SPLINE
SPL {X  -165.650, Y  +556.469, Z    +0.000, E1   +47.823, E3 +319681.375}
SPL {X  -165.650, Y  +549.545, Z    +0.000, E1   +47.953, E3 +319693.501}
SPL {X  -165.650, Y  +541.974, Z    +0.000, E1   +47.882, E3 +319707.890}
SPL {X  -165.650, Y  +535.023, Z    +0.000, E1   +47.697, E3 +319721.879}
SPL {X  -165.650, Y  +526.169, Z    +0.000, E1   +47.853, E3 +319737.474}
SPL {X  -165.650, Y  +520.016, Z    +0.000, E1   +47.658, E3 +319749.858}
SPL {X  -165.650, Y  +512.416, Z    +0.000, E1   +48.035, E3 +319761.825}
SPL {X  -165.650, Y  +507.257, Z    +0.000, E1   +47.748, E3 +319772.892}
SPL {X  -165.650, Y  +501.812, Z    +0.000, E1   +47.738, E3 +319783.175}
SPL {X  -165.650, Y  +493.465, Z    +0.000, E1   +47.959, E3 +319797.346}
SPL {X  -165.650, Y  +486.149, Z    +0.000, E1   +47.831, E3 +319811.621}
SPL {X  -165.650, Y  +479.821, Z    +0.000, E1   +47.727, E3 +319823.895}
SPL {X  -165.650, Y  +472.739, Z    +0.000, E1   +47.923, E3 +319835.914}
SPL {X  -165.650, Y  +466.586, Z    +0.000, E1   +48.125, E3 +319845.928}
SPL {X  -165.650, Y  +464.575, Z    +0.000, E1   +47.451, E3 +319853.694}
SPL {X  -165.650, Y  +456.851, Z    +0.000, E1   +47.856, E3 +319865.800}
SPL {X  -165.650, Y  +449.262, Z    +0.000, E1   +48.080, E3 +319878.366}
SPL {X  -165.650, Y  +436.765, Z    +0.000, E1   +49.819, E3 +319890.265}
SPL {X  -165.650, Y  +430.891, Z    +0.000, E1   +49.130, E3 +319904.767}
SPL {X  -165.650, Y  +423.272, Z    +0.000, E1   +49.176, E3 +319917.805}
SPL {X  -165.650, Y  +416.522, Z    +0.000, E1   +49.338, E3 +319928.783}
SPL {X  -165.650, Y  +410.777, Z    +0.000, E1   +49.173, E3 +319939.835}
SPL {X  -165.650, Y  +405.230, Z    +0.000, E1   +49.266, E3 +319949.038}
SPL {X  -165.650, Y  +398.850, Z    +0.000, E1   +49.279, E3 +319960.330}
SPL {X  -165.650, Y  +391.803, Z    +0.000, E1   +49.319, E3 +319972.367}
SPL {X  -165.650, Y  +386.526, Z    +0.000, E1   +49.193, E3 +319982.457}
SPL {X  -165.650, Y  +381.684, Z    +0.000, E1   +49.061, E3 +319991.742}
SPL {X  -165.602, Y  +374.507, Z    +0.000, E1   +49.269, E3 +320003.334}
SPL {X  -165.183, Y  +366.070, Z    +0.000, E1   +49.261, E3 +320018.218}
SPL {X  -164.692, Y  +360.715, Z    +0.000, E1   +48.960, E3 +320029.299}
SPL {X  -163.908, Y  +354.543, Z    +0.000, E1   +49.169, E3 +320038.990}
SPL {X  -163.052, Y  +349.277, Z    +0.000, E1   +48.680, E3 +320051.095}
SPL {X  -162.125, Y  +344.507, Z    +0.000, E1   +48.543, E3 +320060.235}
SPL {X  -160.947, Y  +339.310, Z    +0.000, E1   +48.561, E3 +320069.344}
SPL {X  -159.860, Y  +335.086, Z    +0.000, E1   +48.145, E3 +320079.056}
SPL {X  -158.277, Y  +329.631, Z    +0.000, E1   +47.981, E3 +320089.678}
SPL {X  -156.804, Y  +325.092, Z    +0.000, E1   +47.609, E3 +320099.571}
SPL {X  -155.465, Y  +321.311, Z    +0.000, E1   +47.446, E3 +320107.106}
SPL {X  -153.706, Y  +316.739, Z    +0.000, E1   +47.523, E3 +320114.719}
SPL {X  -143.727, Y  +296.145, Z    +0.000, E1   +53.260, E3 +320117.863}
SPL {X  -128.440, Y  +273.891, Z    +0.000, E1   +47.966, E3 +320205.109}
ENDSPLINE

SPLINE
SPL {X  -131.798, Y  +278.155, Z    +0.000, E1   +45.574, E3 +320230.736}
SPL {X  -154.181, Y  +317.936, Z    +0.000, E1   +32.662, E3 +320296.072}
SPL {X  -162.537, Y  +346.536, Z    +0.000, E1   +20.123, E3 +320295.293}
SPL {X  -164.610, Y  +359.970, Z    +0.000, E1   +13.118, E3 +320290.159}
SPL {X  -165.367, Y  +368.828, Z    +0.000, E1    +8.137, E3 +320288.612}
SPL {X  -165.621, Y  +375.422, Z    +0.000, E1    +4.067, E3 +320289.489}
SPL {X  -165.650, Y  +379.733, Z    +0.000, E1    +1.160, E3 +320287.795}
SPL {X  -165.650, Y  +383.552, Z    +0.000, E1    -1.868, E3 +320287.045}
SPL {X  -165.650, Y  +387.323, Z    +0.000, E1    -5.609, E3 +320286.861}
SPL {X  -165.650, Y  +392.013, Z    +0.000, E1   -10.856, E3 +320285.878}
SPL {X  -165.650, Y  +398.769, Z    +0.000, E1   -19.304, E3 +320284.490}
SPL {X  -165.650, Y  +407.471, Z    +0.000, E1   -31.017, E3 +320280.648}
SPL {X  -165.650, Y  +414.706, Z    +0.000, E1   -39.242, E3 +320279.624}
SPL {X  -165.650, Y  +446.037, Z    +0.000, E1   -53.739, E3 +320294.230}
SPL {X  -165.650, Y  +454.158, Z    +0.000, E1   -53.343, E3 +320304.582}
SPL {X  -165.650, Y  +513.780, Z    +0.000, E1   -56.183, E3 +320365.379}
ENDSPLINE

SPLINE
SPL {X  -165.650, Y  +495.869, Z    +0.000, E1   -48.812, E3 +320381.567}
ENDSPLINE

SPLINE
SPL {X  -165.650, Y  +504.906, Z    +0.000, E1   -48.979, E3 +320396.887}
SPL {X  -165.650, Y  +512.952, Z    +0.000, E1   -48.898, E3 +320411.509}
SPL {X  -165.650, Y  +519.321, Z    +0.000, E1   -49.041, E3 +320421.977}
SPL {X  -165.650, Y  +524.312, Z    +0.000, E1   -48.855, E3 +320432.002}
SPL {X  -165.650, Y  +530.631, Z    +0.000, E1   -48.990, E3 +320442.462}
SPL {X  -165.650, Y  +536.725, Z    +0.000, E1   -48.843, E3 +320454.213}
SPL {X  -165.650, Y  +542.959, Z    +0.000, E1   -48.923, E3 +320464.828}
SPL {X  -165.650, Y  +548.939, Z    +0.000, E1   -48.968, E3 +320475.222}
SPL {X  -165.650, Y  +553.607, Z    +0.000, E1   -48.716, E3 +320485.040}
SPL {X  -165.650, Y  +562.368, Z    +0.000, E1   -49.014, E3 +320499.100}
SPL {X  -165.650, Y  +570.317, Z    +0.000, E1   -48.893, E3 +320513.843}
SPL {X  -165.650, Y  +577.487, Z    +0.000, E1   -49.001, E3 +320525.951}
SPL {X  -165.650, Y  +581.837, Z    +0.000, E1   -48.612, E3 +320535.984}
SPL {X  -165.650, Y  +588.614, Z    +0.000, E1   -49.053, E3 +320545.502}
SPL {X  -165.650, Y  +593.784, Z    +0.000, E1   -48.711, E3 +320556.787}
SPL {X  -165.650, Y  +600.281, Z    +0.000, E1   -48.957, E3 +320566.890}
SPL {X  -165.650, Y  +606.252, Z    +0.000, E1   -48.984, E3 +320577.423}
SPL {X  -165.650, Y  +612.690, Z    +0.000, E1   -49.044, E3 +320588.452}
SPL {X  -165.650, Y  +617.274, Z    +0.000, E1   -48.670, E3 +320598.901}
SPL {X  -165.650, Y  +624.267, Z    +0.000, E1   -48.953, E3 +320609.713}
SPL {X  -165.650, Y  +632.510, Z    +0.000, E1   -48.976, E3 +320624.467}
SPL {X  -165.650, Y  +641.084, Z    +0.000, E1   -48.892, E3 +320640.110}
SPL {X  -165.650, Y  +648.143, Z    +0.000, E1   -49.033, E3 +320651.779}
SPL {X  -165.650, Y  +655.847, Z    +0.000, E1   -48.917, E3 +320666.397}
SPL {X  -165.650, Y  +663.676, Z    +0.000, E1   -48.809, E3 +320680.835}
SPL {X  -165.650, Y  +669.580, Z    +0.000, E1   -48.844, E3 +320691.173}
SPL {X  -165.650, Y  +675.734, Z    +0.000, E1   -49.021, E3 +320701.079}
SPL {X  -165.552, Y  +681.198, Z    +0.000, E1   -48.804, E3 +320712.160}
SPL {X  -165.221, Y  +687.413, Z    +0.000, E1   -48.790, E3 +320723.331}
SPL {X  -164.785, Y  +692.407, Z    +0.000, E1   -48.653, E3 +320733.047}
SPL {X  -164.074, Y  +698.293, Z    +0.000, E1   -48.857, E3 +320742.331}
SPL {X  -163.489, Y  +702.172, Z    +0.000, E1   -48.443, E3 +320751.648}
SPL {X  -162.671, Y  +706.776, Z    +0.000, E1   -48.273, E3 +320760.867}
SPL {X  -161.177, Y  +713.734, Z    +0.000, E1   -48.156, E3 +320774.153}
SPL {X  -159.392, Y  +720.602, Z    +0.000, E1   -47.892, E3 +320787.707}
SPL {X  -157.947, Y  +725.428, Z    +0.000, E1   -47.498, E3 +320798.446}
SPL {X  -156.133, Y  +730.838, Z    +0.000, E1   -47.305, E3 +320809.163}
SPL {X  -153.862, Y  +736.871, Z    +0.000, E1   -47.425, E3 +320819.149}
SPL {X  -143.211, Y  +758.749, Z    +0.000, E1   -53.445, E3 +320822.793}
SPL {X  -129.526, Y  +778.761, Z    +0.000, E1   -47.396, E3 +320913.535}
ENDSPLINE

SPLINE
SPL {X  -152.848, Y  +739.355, Z    +0.000, E1   -33.672, E3 +320989.104}
SPL {X  -162.700, Y  +706.622, Z    +0.000, E1   -19.657, E3 +320995.260}
SPL {X  -164.822, Y  +692.043, Z    +0.000, E1   -12.043, E3 +320990.899}
SPL {X  -165.501, Y  +682.513, Z    +0.000, E1    -6.586, E3 +320989.593}
SPL {X  -165.650, Y  +674.436, Z    +0.000, E1    -1.443, E3 +320988.369}
SPL {X  -165.650, Y  +670.475, Z    +0.000, E1    +1.794, E3 +320988.030}
SPL {X  -165.650, Y  +667.655, Z    +0.000, E1    +4.420, E3 +320987.826}
SPL {X  -165.650, Y  +663.208, Z    +0.000, E1    +9.118, E3 +320987.008}
SPL {X  -165.650, Y  +657.399, Z    +0.000, E1   +16.251, E3 +320985.127}
SPL {X  -165.650, Y  +650.683, Z    +0.000, E1   +24.801, E3 +320983.102}
SPL {X  -165.650, Y  +636.402, Z    +0.000, E1   +39.824, E3 +320983.065}
SPL {X  -165.650, Y  +586.376, Z    +0.000, E1   +59.481, E3 +321000.737}
SPL {X  -165.650, Y  +554.310, Z    +0.000, E1   +51.914, E3 +321068.781}
ENDSPLINE

SPLINE
SPL {X  -165.650, Y  +561.648, Z    +0.000, E1   +48.058, E3 +321079.598}
ENDSPLINE

SPLINE
SPL {X  -165.650, Y  +556.469, Z    +0.000, E1   +47.823, E3 +321090.466}
SPL {X  -165.650, Y  +549.545, Z    +0.000, E1   +47.953, E3 +321102.592}
SPL {X  -165.650, Y  +541.974, Z    +0.000, E1   +47.882, E3 +321116.981}
SPL {X  -165.650, Y  +535.023, Z    +0.000, E1   +47.697, E3 +321130.970}
SPL {X  -165.650, Y  +526.169, Z    +0.000, E1   +47.853, E3 +321146.565}
SPL {X  -165.650, Y  +517.493, Z    +0.000, E1   +47.895, E3 +321162.312}
SPL {X  -165.650, Y  +509.413, Z    +0.000, E1   +47.884, E3 +321177.391}
SPL {X  -165.650, Y  +501.812, Z    +0.000, E1   +47.738, E3 +321192.266}
SPL {X  -165.650, Y  +494.522, Z    +0.000, E1   +48.055, E3 +321203.793}
SPL {X  -165.650, Y  +489.529, Z    +0.000, E1   +47.849, E3 +321214.247}
SPL {X  -165.650, Y  +481.894, Z    +0.000, E1   +47.756, E3 +321229.148}
SPL {X  -165.650, Y  +472.739, Z    +0.000, E1   +47.923, E3 +321245.005}
SPL {X  -165.650, Y  +466.586, Z    +0.000, E1   +48.125, E3 +321255.019}
SPL {X  -165.650, Y  +464.575, Z    +0.000, E1   +47.451, E3 +321262.785}
SPL {X  -165.650, Y  +457.811, Z    +0.000, E1   +47.987, E3 +321272.201}
SPL {X  -165.650, Y  +451.187, Z    +0.000, E1   +47.917, E3 +321284.945}
SPL {X  -165.650, Y  +436.454, Z    +0.000, E1   +49.483, E3 +321302.164}
SPL {X  -165.650, Y  +428.379, Z    +0.000, E1   +49.373, E3 +321316.760}
SPL {X  -165.650, Y  +423.272, Z    +0.000, E1   +49.176, E3 +321326.896}
SPL {X  -165.650, Y  +416.522, Z    +0.000, E1   +49.338, E3 +321337.874}
SPL {X  -165.650, Y  +408.142, Z    +0.000, E1   +49.261, E3 +321353.235}
SPL {X  -165.650, Y  +400.266, Z    +0.000, E1   +49.362, E3 +321366.296}
SPL {X  -165.650, Y  +393.708, Z    +0.000, E1   +49.252, E3 +321378.602}
SPL {X  -165.650, Y  +384.475, Z    +0.000, E1   +49.187, E3 +321395.401}
SPL {X  -165.602, Y  +374.507, Z    +0.000, E1   +49.269, E3 +321412.425}
SPL {X  -165.183, Y  +366.070, Z    +0.000, E1   +49.261, E3 +321427.309}
SPL {X  -164.692, Y  +360.715, Z    +0.000, E1   +48.960, E3 +321438.390}
SPL {X  -163.908, Y  +354.543, Z    +0.000, E1   +49.169, E3 +321448.081}
SPL {X  -163.052, Y  +349.277, Z    +0.000, E1   +48.680, E3 +321460.186}
SPL {X  -162.125, Y  +344.507, Z    +0.000, E1   +48.543, E3 +321469.326}
SPL {X  -160.947, Y  +339.310, Z    +0.000, E1   +48.561, E3 +321478.435}
SPL {X  -159.499, Y  +333.778, Z    +0.000, E1   +48.145, E3 +321490.547}
SPL {X  -157.957, Y  +328.606, Z    +0.000, E1   +47.890, E3 +321500.972}
SPL {X  -156.095, Y  +323.055, Z    +0.000, E1   +47.566, E3 +321512.656}
SPL {X  -153.706, Y  +316.739, Z    +0.000, E1   +47.523, E3 +321523.810}
SPL {X  -146.106, Y  +300.443, Z    +0.000, E1   +52.765, E3 +321523.429}
SPL {X  -140.816, Y  +291.260, Z    +0.000, E1   +53.766, E3 +321531.112}
SPL {X  -128.440, Y  +273.891, Z    +0.000, E1   +47.966, E3 +321614.200}
ENDSPLINE

SPLINE
SPL {X  -131.798, Y  +278.155, Z    +0.000, E1   +45.574, E3 +321639.827}
SPL {X  -154.181, Y  +317.936, Z    +0.000, E1   +32.662, E3 +321705.163}
SPL {X  -162.537, Y  +346.536, Z    +0.000, E1   +20.123, E3 +321704.384}
SPL {X  -165.197, Y  +366.255, Z    +0.000, E1    +9.700, E3 +321698.179}
SPL {X  -165.621, Y  +375.422, Z    +0.000, E1    +4.067, E3 +321698.580}
SPL {X  -165.650, Y  +379.733, Z    +0.000, E1    +1.160, E3 +321696.886}
SPL {X  -165.650, Y  +383.552, Z    +0.000, E1    -1.868, E3 +321696.135}
SPL {X  -165.650, Y  +387.323, Z    +0.000, E1    -5.609, E3 +321695.952}
SPL {X  -165.650, Y  +392.013, Z    +0.000, E1   -10.856, E3 +321694.969}
SPL {X  -165.650, Y  +398.769, Z    +0.000, E1   -19.304, E3 +321693.580}
SPL {X  -165.650, Y  +410.885, Z    +0.000, E1   -34.864, E3 +321689.257}
SPL {X  -165.650, Y  +448.279, Z    +0.000, E1   -53.294, E3 +321707.102}
SPL {X  -165.650, Y  +465.286, Z    +0.000, E1   -55.209, E3 +321720.953}
SPL {X  -165.650, Y  +513.874, Z    +0.000, E1   -57.683, E3 +321765.762}
ENDSPLINE

SPLINE
SPL {X  -165.650, Y  +513.412, Z    +0.000, E1   -55.245, E3 +321779.357}
SPL {X  -165.650, Y  +495.869, Z    +0.000, E1   -48.812, E3 +321790.658}
ENDSPLINE

SPLINE
SPL {X  -165.650, Y  +502.040, Z    +0.000, E1   -48.856, E3 +321801.402}
SPL {X  -165.650, Y  +507.863, Z    +0.000, E1   -49.013, E3 +321810.822}
SPL {X  -165.650, Y  +512.952, Z    +0.000, E1   -48.898, E3 +321820.599}
SPL {X  -165.650, Y  +519.321, Z    +0.000, E1   -49.041, E3 +321831.067}
SPL {X  -165.650, Y  +524.312, Z    +0.000, E1   -48.855, E3 +321841.093}
SPL {X  -165.650, Y  +530.631, Z    +0.000, E1   -48.990, E3 +321851.553}
SPL {X  -165.650, Y  +536.725, Z    +0.000, E1   -48.843, E3 +321863.304}
SPL {X  -165.650, Y  +542.959, Z    +0.000, E1   -48.923, E3 +321873.919}
SPL {X  -165.650, Y  +548.939, Z    +0.000, E1   -48.968, E3 +321884.312}
SPL {X  -165.650, Y  +553.607, Z    +0.000, E1   -48.716, E3 +321894.130}
SPL {X  -165.650, Y  +562.368, Z    +0.000, E1   -49.014, E3 +321908.191}
SPL {X  -165.650, Y  +570.317, Z    +0.000, E1   -48.893, E3 +321922.933}
SPL {X  -165.650, Y  +577.487, Z    +0.000, E1   -49.001, E3 +321935.042}
SPL {X  -165.650, Y  +581.837, Z    +0.000, E1   -48.612, E3 +321945.075}
SPL {X  -165.650, Y  +588.614, Z    +0.000, E1   -49.053, E3 +321954.593}
SPL {X  -165.650, Y  +593.784, Z    +0.000, E1   -48.711, E3 +321965.878}
SPL {X  -165.650, Y  +600.281, Z    +0.000, E1   -48.957, E3 +321975.981}
SPL {X  -165.650, Y  +606.252, Z    +0.000, E1   -48.984, E3 +321986.514}
SPL {X  -165.650, Y  +612.690, Z    +0.000, E1   -49.044, E3 +321997.543}
SPL {X  -165.650, Y  +617.274, Z    +0.000, E1   -48.670, E3 +322007.992}
SPL {X  -165.650, Y  +624.267, Z    +0.000, E1   -48.953, E3 +322018.804}
SPL {X  -165.650, Y  +632.510, Z    +0.000, E1   -48.976, E3 +322033.558}
SPL {X  -165.650, Y  +641.084, Z    +0.000, E1   -48.892, E3 +322049.201}
SPL {X  -165.650, Y  +648.143, Z    +0.000, E1   -49.033, E3 +322060.870}
SPL {X  -165.650, Y  +652.108, Z    +0.000, E1   -48.593, E3 +322070.555}
SPL {X  -165.650, Y  +658.753, Z    +0.000, E1   -49.107, E3 +322079.380}
SPL {X  -165.650, Y  +663.676, Z    +0.000, E1   -48.809, E3 +322089.925}
SPL {X  -165.650, Y  +669.580, Z    +0.000, E1   -48.844, E3 +322100.264}
SPL {X  -165.650, Y  +675.734, Z    +0.000, E1   -49.021, E3 +322110.170}
SPL {X  -165.552, Y  +681.198, Z    +0.000, E1   -48.804, E3 +322121.251}
SPL {X  -165.221, Y  +687.413, Z    +0.000, E1   -48.790, E3 +322132.422}
SPL {X  -164.785, Y  +692.407, Z    +0.000, E1   -48.653, E3 +322142.138}
SPL {X  -164.074, Y  +698.293, Z    +0.000, E1   -48.857, E3 +322151.422}
SPL {X  -163.489, Y  +702.172, Z    +0.000, E1   -48.443, E3 +322160.739}
SPL {X  -162.217, Y  +709.048, Z    +0.000, E1   -48.328, E3 +322173.878}
SPL {X  -160.800, Y  +715.289, Z    +0.000, E1   -47.964, E3 +322186.886}
SPL {X  -159.392, Y  +720.602, Z    +0.000, E1   -47.892, E3 +322196.798}
SPL {X  -157.947, Y  +725.428, Z    +0.000, E1   -47.498, E3 +322207.537}
SPL {X  -156.133, Y  +730.838, Z    +0.000, E1   -47.305, E3 +322218.254}
SPL {X  -154.870, Y  +734.280, Z    +0.000, E1   -46.924, E3 +322226.257}
SPL {X  -150.529, Y  +744.645, Z    +0.000, E1   -49.720, E3 +322229.531}
SPL {X  -140.987, Y  +762.463, Z    +0.000, E1   -53.922, E3 +322234.562}
SPL {X  -130.133, Y  +777.996, Z    +0.000, E1   -46.969, E3 +322326.987}
ENDSPLINE

SPLINE
SPL {X  -153.839, Y  +736.929, Z    +0.000, E1   -32.772, E3 +322400.058}
SPL {X  -162.700, Y  +706.622, Z    +0.000, E1   -19.657, E3 +322404.351}
SPL {X  -164.822, Y  +692.043, Z    +0.000, E1   -12.043, E3 +322399.990}
SPL {X  -165.501, Y  +682.513, Z    +0.000, E1    -6.586, E3 +322398.684}
SPL {X  -165.645, Y  +676.829, Z    +0.000, E1    -2.974, E3 +322398.028}
SPL {X  -165.650, Y  +673.338, Z    +0.000, E1    -0.547, E3 +322397.197}
SPL {X  -165.650, Y  +670.475, Z    +0.000, E1    +1.794, E3 +322397.121}
SPL {X  -165.650, Y  +667.655, Z    +0.000, E1    +4.420, E3 +322396.917}
SPL {X  -165.650, Y  +664.048, Z    +0.000, E1    +8.230, E3 +322396.294}
SPL {X  -165.650, Y  +658.867, Z    +0.000, E1   +14.313, E3 +322394.757}
SPL {X  -165.650, Y  +650.683, Z    +0.000, E1   +24.801, E3 +322392.193}
SPL {X  -165.650, Y  +640.858, Z    +0.000, E1   +34.904, E3 +322393.936}
SPL {X  -165.650, Y  +633.111, Z    +0.000, E1   +43.522, E3 +322390.830}
SPL {X  -165.650, Y  +594.935, Z    +0.000, E1   +58.150, E3 +322405.430}
SPL {X  -165.650, Y  +579.579, Z    +0.000, E1   +60.394, E3 +322413.315}
SPL {X  -165.650, Y  +536.483, Z    +0.000, E1   +57.139, E3 +322471.596}
ENDSPLINE

SPLINE
SPL {X  -165.650, Y  +561.248, Z    +0.000, E1   +49.247, E3 +322482.287}
ENDSPLINE

SPLINE
SPL {X  -165.650, Y  +558.330, Z    +0.000, E1   +47.867, E3 +322496.011}
SPL {X  -165.650, Y  +550.626, Z    +0.000, E1   +48.045, E3 +322509.021}
SPL {X  -165.650, Y  +545.464, Z    +0.000, E1   +47.668, E3 +322520.889}
SPL {X  -165.650, Y  +535.912, Z    +0.000, E1   +47.888, E3 +322537.475}
SPL {X  -165.650, Y  +526.169, Z    +0.000, E1   +47.853, E3 +322555.656}
SPL {X  -165.650, Y  +517.493, Z    +0.000, E1   +47.895, E3 +322571.403}
SPL {X  -165.650, Y  +511.255, Z    +0.000, E1   +47.920, E3 +322582.692}
SPL {X  -165.650, Y  +507.257, Z    +0.000, E1   +47.748, E3 +322591.074}
SPL {X  -165.650, Y  +501.812, Z    +0.000, E1   +47.738, E3 +322601.357}
SPL {X  -165.650, Y  +494.522, Z    +0.000, E1   +48.055, E3 +322612.884}
SPL {X  -165.650, Y  +489.529, Z    +0.000, E1   +47.849, E3 +322623.338}
SPL {X  -165.650, Y  +484.859, Z    +0.000, E1   +47.688, E3 +322632.908}
SPL {X  -165.650, Y  +477.718, Z    +0.000, E1   +47.870, E3 +322645.242}
SPL {X  -165.650, Y  +469.088, Z    +0.000, E1   +47.982, E3 +322660.461}
SPL {X  -165.650, Y  +464.575, Z    +0.000, E1   +47.451, E3 +322671.876}
SPL {X  -165.650, Y  +456.851, Z    +0.000, E1   +47.856, E3 +322683.982}
SPL {X  -165.650, Y  +449.262, Z    +0.000, E1   +48.080, E3 +322696.548}
SPL {X  -165.650, Y  +436.765, Z    +0.000, E1   +49.819, E3 +322708.446}
SPL {X  -165.650, Y  +430.891, Z    +0.000, E1   +49.130, E3 +322722.949}
SPL {X  -165.650, Y  +423.272, Z    +0.000, E1   +49.176, E3 +322735.987}
SPL {X  -165.650, Y  +416.522, Z    +0.000, E1   +49.338, E3 +322746.964}
SPL {X  -165.650, Y  +408.142, Z    +0.000, E1   +49.261, E3 +322762.326}
SPL {X  -165.650, Y  +400.266, Z    +0.000, E1   +49.362, E3 +322775.387}
SPL {X  -165.650, Y  +393.708, Z    +0.000, E1   +49.252, E3 +322787.693}
SPL {X  -165.650, Y  +384.475, Z    +0.000, E1   +49.187, E3 +322804.492}
SPL {X  -165.626, Y  +375.686, Z    +0.000, E1   +49.367, E3 +322818.709}
SPL {X  -165.370, Y  +368.879, Z    +0.000, E1   +49.286, E3 +322831.263}
SPL {X  -164.828, Y  +362.023, Z    +0.000, E1   +48.964, E3 +322845.224}
SPL {X  -163.908, Y  +354.543, Z    +0.000, E1   +49.169, E3 +322857.171}
SPL {X  -163.052, Y  +349.277, Z    +0.000, E1   +48.680, E3 +322869.277}
SPL {X  -162.125, Y  +344.507, Z    +0.000, E1   +48.543, E3 +322878.417}
SPL {X  -160.947, Y  +339.310, Z    +0.000, E1   +48.561, E3 +322887.526}
SPL {X  -159.499, Y  +333.778, Z    +0.000, E1   +48.145, E3 +322899.638}
SPL {X  -157.957, Y  +328.606, Z    +0.000, E1   +47.890, E3 +322910.063}
SPL {X  -156.095, Y  +323.055, Z    +0.000, E1   +47.566, E3 +322921.747}
SPL {X  -153.706, Y  +316.739, Z    +0.000, E1   +47.523, E3 +322932.901}
SPL {X  -143.727, Y  +296.145, Z    +0.000, E1   +53.260, E3 +322936.045}
SPL {X  -128.440, Y  +273.891, Z    +0.000, E1   +47.966, E3 +323023.291}
ENDSPLINE

SPLINE
SPL {X  -131.798, Y  +278.155, Z    +0.000, E1   +45.574, E3 +323048.918}
SPL {X  -154.181, Y  +317.936, Z    +0.000, E1   +32.662, E3 +323114.254}
SPL {X  -162.537, Y  +346.536, Z    +0.000, E1   +20.123, E3 +323113.475}
SPL {X  -165.197, Y  +366.255, Z    +0.000, E1    +9.700, E3 +323107.270}
SPL {X  -165.621, Y  +375.422, Z    +0.000, E1    +4.067, E3 +323107.671}
SPL {X  -165.650, Y  +379.733, Z    +0.000, E1    +1.160, E3 +323105.977}
SPL {X  -165.650, Y  +383.552, Z    +0.000, E1    -1.868, E3 +323105.226}
SPL {X  -165.650, Y  +388.716, Z    +0.000, E1    -7.003, E3 +323104.631}
SPL {X  -165.650, Y  +396.644, Z    +0.000, E1   -16.434, E3 +323103.250}
SPL {X  -165.650, Y  +410.885, Z    +0.000, E1   -34.864, E3 +323098.348}
SPL {X  -165.650, Y  +446.037, Z    +0.000, E1   -53.739, E3 +323112.412}
SPL {X  -165.650, Y  +454.158, Z    +0.000, E1   -53.343, E3 +323122.764}
SPL {X  -165.650, Y  +513.780, Z    +0.000, E1   -56.183, E3 +323183.561}
ENDSPLINE

SPLINE
SPL {X  -165.650, Y  +495.869, Z    +0.000, E1   -48.812, E3 +323199.749}
ENDSPLINE

SPLINE
SPL {X  -165.650, Y  +502.040, Z    +0.000, E1   -48.856, E3 +323210.493}
SPL {X  -165.650, Y  +507.863, Z    +0.000, E1   -49.013, E3 +323219.913}
SPL {X  -165.650, Y  +512.952, Z    +0.000, E1   -48.898, E3 +323229.690}
SPL {X  -165.650, Y  +519.321, Z    +0.000, E1   -49.041, E3 +323240.158}
SPL {X  -165.650, Y  +524.312, Z    +0.000, E1   -48.855, E3 +323250.184}
SPL {X  -165.650, Y  +530.631, Z    +0.000, E1   -48.990, E3 +323260.644}
SPL {X  -165.650, Y  +536.725, Z    +0.000, E1   -48.843, E3 +323272.395}
SPL {X  -165.650, Y  +542.959, Z    +0.000, E1   -48.923, E3 +323283.010}
SPL {X  -165.650, Y  +548.939, Z    +0.000, E1   -48.968, E3 +323293.403}
SPL {X  -165.650, Y  +553.607, Z    +0.000, E1   -48.716, E3 +323303.221}
SPL {X  -165.650, Y  +562.368, Z    +0.000, E1   -49.014, E3 +323317.282}
SPL {X  -165.650, Y  +570.317, Z    +0.000, E1   -48.893, E3 +323332.024}
SPL {X  -165.650, Y  +577.487, Z    +0.000, E1   -49.001, E3 +323344.132}
SPL {X  -165.650, Y  +581.837, Z    +0.000, E1   -48.612, E3 +323354.166}
SPL {X  -165.650, Y  +588.614, Z    +0.000, E1   -49.053, E3 +323363.684}
SPL {X  -165.650, Y  +593.784, Z    +0.000, E1   -48.711, E3 +323374.969}
SPL {X  -165.650, Y  +600.281, Z    +0.000, E1   -48.957, E3 +323385.072}
SPL {X  -165.650, Y  +606.252, Z    +0.000, E1   -48.984, E3 +323395.605}
SPL {X  -165.650, Y  +612.690, Z    +0.000, E1   -49.044, E3 +323406.634}
SPL {X  -165.650, Y  +617.274, Z    +0.000, E1   -48.670, E3 +323417.083}
SPL {X  -165.650, Y  +624.267, Z    +0.000, E1   -48.953, E3 +323427.895}
SPL {X  -165.650, Y  +632.510, Z    +0.000, E1   -48.976, E3 +323442.649}
SPL {X  -165.650, Y  +641.084, Z    +0.000, E1   -48.892, E3 +323458.292}
SPL {X  -165.650, Y  +648.143, Z    +0.000, E1   -49.033, E3 +323469.961}
SPL {X  -165.650, Y  +652.108, Z    +0.000, E1   -48.593, E3 +323479.645}
SPL {X  -165.650, Y  +658.753, Z    +0.000, E1   -49.107, E3 +323488.471}
SPL {X  -165.650, Y  +663.676, Z    +0.000, E1   -48.809, E3 +323499.016}
SPL {X  -165.650, Y  +669.580, Z    +0.000, E1   -48.844, E3 +323509.355}
SPL {X  -165.650, Y  +675.734, Z    +0.000, E1   -49.021, E3 +323519.261}
SPL {X  -165.552, Y  +681.198, Z    +0.000, E1   -48.804, E3 +323530.341}
SPL {X  -165.221, Y  +687.413, Z    +0.000, E1   -48.790, E3 +323541.513}
SPL {X  -164.785, Y  +692.407, Z    +0.000, E1   -48.653, E3 +323551.229}
SPL {X  -164.074, Y  +698.293, Z    +0.000, E1   -48.857, E3 +323560.513}
SPL {X  -163.489, Y  +702.172, Z    +0.000, E1   -48.443, E3 +323569.829}
SPL {X  -162.217, Y  +709.048, Z    +0.000, E1   -48.328, E3 +323582.969}
SPL {X  -160.800, Y  +715.289, Z    +0.000, E1   -47.964, E3 +323595.977}
SPL {X  -159.392, Y  +720.602, Z    +0.000, E1   -47.892, E3 +323605.889}
SPL {X  -157.947, Y  +725.428, Z    +0.000, E1   -47.498, E3 +323616.628}
SPL {X  -155.696, Y  +732.057, Z    +0.000, E1   -47.224, E3 +323630.104}
SPL {X  -152.475, Y  +740.240, Z    +0.000, E1   -48.059, E3 +323639.934}
SPL {X  -143.211, Y  +758.749, Z    +0.000, E1   -53.445, E3 +323640.975}
SPL {X  -129.526, Y  +778.761, Z    +0.000, E1   -47.396, E3 +323731.717}
ENDSPLINE

SPLINE
SPL {X  -152.848, Y  +739.355, Z    +0.000, E1   -33.672, E3 +323807.286}
SPL {X  -162.700, Y  +706.622, Z    +0.000, E1   -19.657, E3 +323813.442}
SPL {X  -164.822, Y  +692.043, Z    +0.000, E1   -12.043, E3 +323809.081}
SPL {X  -165.501, Y  +682.513, Z    +0.000, E1    -6.586, E3 +323807.775}
SPL {X  -165.650, Y  +674.436, Z    +0.000, E1    -1.443, E3 +323806.551}
SPL {X  -165.650, Y  +669.008, Z    +0.000, E1    +2.993, E3 +323806.106}
SPL {X  -165.650, Y  +664.048, Z    +0.000, E1    +8.230, E3 +323805.384}
SPL {X  -165.650, Y  +658.867, Z    +0.000, E1   +14.313, E3 +323803.848}
SPL {X  -165.650, Y  +650.683, Z    +0.000, E1   +24.801, E3 +323801.284}
SPL {X  -165.650, Y  +640.858, Z    +0.000, E1   +34.904, E3 +323803.027}
SPL {X  -165.650, Y  +633.111, Z    +0.000, E1   +43.522, E3 +323799.921}
SPL {X  -165.650, Y  +586.376, Z    +0.000, E1   +59.481, E3 +323818.919}
SPL {X  -165.650, Y  +554.310, Z    +0.000, E1   +51.914, E3 +323886.963}
ENDSPLINE

SPLINE
SPL {X  -165.650, Y  +561.648, Z    +0.000, E1   +48.058, E3 +323897.780}
ENDSPLINE

SPLINE
SPL {X  -165.650, Y  +556.469, Z    +0.000, E1   +47.823, E3 +323908.648}
SPL {X  -165.650, Y  +549.545, Z    +0.000, E1   +47.953, E3 +323920.774}
SPL {X  -165.650, Y  +541.974, Z    +0.000, E1   +47.882, E3 +323935.163}
SPL {X  -165.650, Y  +535.023, Z    +0.000, E1   +47.697, E3 +323949.152}
SPL {X  -165.650, Y  +526.169, Z    +0.000, E1   +47.853, E3 +323964.746}
SPL {X  -165.650, Y  +520.016, Z    +0.000, E1   +47.658, E3 +323977.131}
SPL {X  -165.650, Y  +512.416, Z    +0.000, E1   +48.035, E3 +323989.098}
SPL {X  -165.650, Y  +507.257, Z    +0.000, E1   +47.748, E3 +324000.165}
SPL {X  -165.650, Y  +501.812, Z    +0.000, E1   +47.738, E3 +324010.448}
SPL {X  -165.650, Y  +494.522, Z    +0.000, E1   +48.055, E3 +324021.975}
SPL {X  -165.650, Y  +489.529, Z    +0.000, E1   +47.849, E3 +324032.429}
SPL {X  -165.650, Y  +484.859, Z    +0.000, E1   +47.688, E3 +324041.999}
SPL {X  -165.650, Y  +477.718, Z    +0.000, E1   +47.870, E3 +324054.333}
SPL {X  -165.650, Y  +469.088, Z    +0.000, E1   +47.982, E3 +324069.552}
SPL {X  -165.650, Y  +464.575, Z    +0.000, E1   +47.451, E3 +324080.967}
SPL {X  -165.650, Y  +456.851, Z    +0.000, E1   +47.856, E3 +324093.073}
SPL {X  -165.650, Y  +449.262, Z    +0.000, E1   +48.080, E3 +324105.639}
SPL {X  -165.650, Y  +436.454, Z    +0.000, E1   +49.483, E3 +324120.345}
SPL {X  -165.650, Y  +428.379, Z    +0.000, E1   +49.373, E3 +324134.942}
SPL {X  -165.650, Y  +423.272, Z    +0.000, E1   +49.176, E3 +324145.078}
SPL {X  -165.650, Y  +416.522, Z    +0.000, E1   +49.338, E3 +324156.055}
SPL {X  -165.650, Y  +410.777, Z    +0.000, E1   +49.173, E3 +324167.108}
SPL {X  -165.650, Y  +405.230, Z    +0.000, E1   +49.266, E3 +324176.311}
SPL {X  -165.650, Y  +398.850, Z    +0.000, E1   +49.279, E3 +324187.603}
SPL {X  -165.650, Y  +391.803, Z    +0.000, E1   +49.319, E3 +324199.640}
SPL {X  -165.650, Y  +386.526, Z    +0.000, E1   +49.193, E3 +324209.730}
SPL {X  -165.649, Y  +378.059, Z    +0.000, E1   +49.283, E3 +324224.272}
SPL {X  -165.292, Y  +367.617, Z    +0.000, E1   +49.239, E3 +324243.038}
SPL {X  -164.692, Y  +360.715, Z    +0.000, E1   +48.960, E3 +324256.572}
SPL {X  -163.908, Y  +354.543, Z    +0.000, E1   +49.169, E3 +324266.262}
SPL {X  -163.052, Y  +349.277, Z    +0.000, E1   +48.680, E3 +324278.368}
SPL {X  -162.125, Y  +344.507, Z    +0.000, E1   +48.543, E3 +324287.508}
SPL {X  -160.947, Y  +339.310, Z    +0.000, E1   +48.561, E3 +324296.617}
SPL {X  -159.860, Y  +335.086, Z    +0.000, E1   +48.145, E3 +324306.329}
SPL {X  -158.277, Y  +329.631, Z    +0.000, E1   +47.981, E3 +324316.951}
SPL {X  -156.095, Y  +323.055, Z    +0.000, E1   +47.566, E3 +324330.838}
SPL {X  -153.706, Y  +316.739, Z    +0.000, E1   +47.523, E3 +324341.992}
SPL {X  -143.727, Y  +296.145, Z    +0.000, E1   +53.260, E3 +324345.135}
SPL {X  -128.440, Y  +273.891, Z    +0.000, E1   +47.966, E3 +324432.382}
ENDSPLINE

SPLINE
SPL {X  -131.798, Y  +278.155, Z    +0.000, E1   +45.574, E3 +324458.009}
SPL {X  -154.181, Y  +317.936, Z    +0.000, E1   +32.662, E3 +324523.345}
SPL {X  -162.537, Y  +346.536, Z    +0.000, E1   +20.123, E3 +324522.566}
SPL {X  -164.610, Y  +359.970, Z    +0.000, E1   +13.118, E3 +324517.432}
SPL {X  -165.367, Y  +368.828, Z    +0.000, E1    +8.137, E3 +324515.885}
SPL {X  -165.621, Y  +375.422, Z    +0.000, E1    +4.067, E3 +324516.762}
SPL {X  -165.650, Y  +379.733, Z    +0.000, E1    +1.160, E3 +324515.068}
SPL {X  -165.650, Y  +383.552, Z    +0.000, E1    -1.868, E3 +324514.317}
SPL {X  -165.650, Y  +387.323, Z    +0.000, E1    -5.609, E3 +324514.134}
SPL {X  -165.650, Y  +392.013, Z    +0.000, E1   -10.856, E3 +324513.151}
SPL {X  -165.650, Y  +398.769, Z    +0.000, E1   -19.304, E3 +324511.762}
SPL {X  -165.650, Y  +410.885, Z    +0.000, E1   -34.864, E3 +324507.438}
SPL {X  -165.650, Y  +448.279, Z    +0.000, E1   -53.294, E3 +324525.283}
SPL {X  -165.650, Y  +465.286, Z    +0.000, E1   -55.209, E3 +324539.135}
SPL {X  -165.650, Y  +513.874, Z    +0.000, E1   -57.683, E3 +324583.944}
ENDSPLINE

SPLINE
SPL {X  -165.650, Y  +513.412, Z    +0.000, E1   -55.245, E3 +324597.539}
SPL {X  -165.650, Y  +495.869, Z    +0.000, E1   -48.812, E3 +324608.840}
ENDSPLINE

SPLINE
SPL {X  -165.650, Y  +502.040, Z    +0.000, E1   -48.856, E3 +324619.584}
SPL {X  -165.650, Y  +507.863, Z    +0.000, E1   -49.013, E3 +324629.004}
SPL {X  -165.650, Y  +512.952, Z    +0.000, E1   -48.898, E3 +324638.781}
SPL {X  -165.650, Y  +519.321, Z    +0.000, E1   -49.041, E3 +324649.249}
SPL {X  -165.650, Y  +524.312, Z    +0.000, E1   -48.855, E3 +324659.275}
SPL {X  -165.650, Y  +530.631, Z    +0.000, E1   -48.990, E3 +324669.735}
SPL {X  -165.650, Y  +536.725, Z    +0.000, E1   -48.843, E3 +324681.485}
SPL {X  -165.650, Y  +542.959, Z    +0.000, E1   -48.923, E3 +324692.100}
SPL {X  -165.650, Y  +548.939, Z    +0.000, E1   -48.968, E3 +324702.494}
SPL {X  -165.650, Y  +553.607, Z    +0.000, E1   -48.716, E3 +324712.312}
SPL {X  -165.650, Y  +560.535, Z    +0.000, E1   -49.121, E3 +324722.261}
SPL {X  -165.650, Y  +564.320, Z    +0.000, E1   -48.789, E3 +324730.949}
SPL {X  -165.650, Y  +570.317, Z    +0.000, E1   -48.893, E3 +324741.115}
SPL {X  -165.650, Y  +577.487, Z    +0.000, E1   -49.001, E3 +324753.223}
SPL {X  -165.650, Y  +581.837, Z    +0.000, E1   -48.612, E3 +324763.257}
SPL {X  -165.650, Y  +588.614, Z    +0.000, E1   -49.053, E3 +324772.775}
SPL {X  -165.650, Y  +593.784, Z    +0.000, E1   -48.711, E3 +324784.060}
SPL {X  -165.650, Y  +600.281, Z    +0.000, E1   -48.957, E3 +324794.163}
SPL {X  -165.650, Y  +606.252, Z    +0.000, E1   -48.984, E3 +324804.696}
SPL {X  -165.650, Y  +612.690, Z    +0.000, E1   -49.044, E3 +324815.725}
SPL {X  -165.650, Y  +617.274, Z    +0.000, E1   -48.670, E3 +324826.174}
SPL {X  -165.650, Y  +624.267, Z    +0.000, E1   -48.953, E3 +324836.986}
SPL {X  -165.650, Y  +632.510, Z    +0.000, E1   -48.976, E3 +324851.740}
SPL {X  -165.650, Y  +641.084, Z    +0.000, E1   -48.892, E3 +324867.383}
SPL {X  -165.650, Y  +648.143, Z    +0.000, E1   -49.033, E3 +324879.052}
SPL {X  -165.650, Y  +655.847, Z    +0.000, E1   -48.917, E3 +324893.669}
SPL {X  -165.650, Y  +663.676, Z    +0.000, E1   -48.809, E3 +324908.107}
SPL {X  -165.650, Y  +669.580, Z    +0.000, E1   -48.844, E3 +324918.446}
SPL {X  -165.650, Y  +675.734, Z    +0.000, E1   -49.021, E3 +324928.352}
SPL {X  -165.552, Y  +681.198, Z    +0.000, E1   -48.804, E3 +324939.432}
SPL {X  -165.221, Y  +687.413, Z    +0.000, E1   -48.790, E3 +324950.604}
SPL {X  -164.785, Y  +692.407, Z    +0.000, E1   -48.653, E3 +324960.320}
SPL {X  -164.074, Y  +698.293, Z    +0.000, E1   -48.857, E3 +324969.604}
SPL {X  -163.489, Y  +702.172, Z    +0.000, E1   -48.443, E3 +324978.920}
SPL {X  -162.217, Y  +709.048, Z    +0.000, E1   -48.328, E3 +324992.060}
SPL {X  -160.800, Y  +715.289, Z    +0.000, E1   -47.964, E3 +325005.068}
SPL {X  -159.392, Y  +720.602, Z    +0.000, E1   -47.892, E3 +325014.980}
SPL {X  -157.947, Y  +725.428, Z    +0.000, E1   -47.498, E3 +325025.719}
SPL {X  -156.133, Y  +730.838, Z    +0.000, E1   -47.305, E3 +325036.435}
SPL {X  -154.870, Y  +734.280, Z    +0.000, E1   -46.924, E3 +325044.439}
SPL {X  -150.529, Y  +744.645, Z    +0.000, E1   -49.720, E3 +325047.713}
SPL {X  -140.987, Y  +762.463, Z    +0.000, E1   -53.922, E3 +325052.744}
SPL {X  -130.133, Y  +777.996, Z    +0.000, E1   -46.969, E3 +325145.169}
ENDSPLINE

SPLINE
SPL {X  -153.839, Y  +736.929, Z    +0.000, E1   -32.772, E3 +325218.240}
SPL {X  -162.700, Y  +706.622, Z    +0.000, E1   -19.657, E3 +325222.533}
SPL {X  -164.822, Y  +692.043, Z    +0.000, E1   -12.043, E3 +325218.172}
SPL {X  -165.501, Y  +682.513, Z    +0.000, E1    -6.586, E3 +325216.866}
SPL {X  -165.645, Y  +676.829, Z    +0.000, E1    -2.974, E3 +325216.210}
SPL {X  -165.650, Y  +673.338, Z    +0.000, E1    -0.547, E3 +325215.379}
SPL {X  -165.650, Y  +669.008, Z    +0.000, E1    +2.993, E3 +325215.196}
SPL {X  -165.650, Y  +664.048, Z    +0.000, E1    +8.230, E3 +325214.475}
SPL {X  -165.650, Y  +658.867, Z    +0.000, E1   +14.313, E3 +325212.939}
SPL {X  -165.650, Y  +650.683, Z    +0.000, E1   +24.801, E3 +325210.375}
SPL {X  -165.650, Y  +636.402, Z    +0.000, E1   +39.824, E3 +325210.337}
SPL {X  -165.650, Y  +586.376, Z    +0.000, E1   +59.481, E3 +325228.010}
SPL {X  -165.650, Y  +536.483, Z    +0.000, E1   +57.139, E3 +325289.778}
ENDSPLINE

SPLINE
SPL {X  -165.650, Y  +560.944, Z    +0.000, E1   +48.666, E3 +325304.800}
ENDSPLINE

SPLINE
SPL {X  -165.650, Y  +556.469, Z    +0.000, E1   +47.823, E3 +325317.739}
SPL {X  -165.650, Y  +550.626, Z    +0.000, E1   +48.045, E3 +325327.203}
SPL {X  -165.650, Y  +545.464, Z    +0.000, E1   +47.668, E3 +325339.071}
SPL {X  -165.650, Y  +537.837, Z    +0.000, E1   +47.880, E3 +325351.949}
SPL {X  -165.650, Y  +530.616, Z    +0.000, E1   +47.886, E3 +325365.314}
SPL {X  -165.650, Y  +522.460, Z    +0.000, E1   +47.738, E3 +325381.424}
SPL {X  -165.650, Y  +512.416, Z    +0.000, E1   +48.035, E3 +325398.189}
SPL {X  -165.650, Y  +507.257, Z    +0.000, E1   +47.748, E3 +325409.256}
SPL {X  -165.650, Y  +501.812, Z    +0.000, E1   +47.738, E3 +325419.539}
SPL {X  -165.650, Y  +494.522, Z    +0.000, E1   +48.055, E3 +325431.066}
SPL {X  -165.650, Y  +489.529, Z    +0.000, E1   +47.849, E3 +325441.519}
SPL {X  -165.650, Y  +481.894, Z    +0.000, E1   +47.756, E3 +325456.421}
SPL {X  -165.650, Y  +472.739, Z    +0.000, E1   +47.923, E3 +325472.277}
SPL {X  -165.650, Y  +466.586, Z    +0.000, E1   +48.125, E3 +325482.292}
SPL {X  -165.650, Y  +464.575, Z    +0.000, E1   +47.451, E3 +325490.058}
SPL {X  -165.650, Y  +457.811, Z    +0.000, E1   +47.987, E3 +325499.474}
SPL {X  -165.650, Y  +451.187, Z    +0.000, E1   +47.917, E3 +325512.217}
SPL {X  -165.650, Y  +436.454, Z    +0.000, E1   +49.483, E3 +325529.436}
SPL {X  -165.650, Y  +428.379, Z    +0.000, E1   +49.373, E3 +325544.033}
SPL {X  -165.650, Y  +423.272, Z    +0.000, E1   +49.176, E3 +325554.169}
SPL {X  -165.650, Y  +416.522, Z    +0.000, E1   +49.338, E3 +325565.146}
SPL {X  -165.650, Y  +408.142, Z    +0.000, E1   +49.261, E3 +325580.507}
SPL {X  -165.650, Y  +400.266, Z    +0.000, E1   +49.362, E3 +325593.569}
SPL {X  -165.650, Y  +393.708, Z    +0.000, E1   +49.252, E3 +325605.875}
SPL {X  -165.650, Y  +384.475, Z    +0.000, E1   +49.187, E3 +325622.674}
SPL {X  -165.602, Y  +374.507, Z    +0.000, E1   +49.269, E3 +325639.697}
SPL {X  -165.183, Y  +366.070, Z    +0.000, E1   +49.261, E3 +325654.582}
SPL {X  -164.692, Y  +360.715, Z    +0.000, E1   +48.960, E3 +325665.663}
SPL {X  -163.908, Y  +354.543, Z    +0.000, E1   +49.169, E3 +325675.353}
SPL {X  -163.052, Y  +349.277, Z    +0.000, E1   +48.680, E3 +325687.459}
SPL {X  -162.125, Y  +344.507, Z    +0.000, E1   +48.543, E3 +325696.599}
SPL {X  -160.947, Y  +339.310, Z    +0.000, E1   +48.561, E3 +325705.708}
SPL {X  -159.499, Y  +333.778, Z    +0.000, E1   +48.145, E3 +325717.820}
SPL {X  -157.957, Y  +328.606, Z    +0.000, E1   +47.890, E3 +325728.245}
SPL {X  -156.095, Y  +323.055, Z    +0.000, E1   +47.566, E3 +325739.929}
SPL {X  -153.706, Y  +316.739, Z    +0.000, E1   +47.523, E3 +325751.083}
SPL {X  -146.106, Y  +300.443, Z    +0.000, E1   +52.765, E3 +325750.702}
SPL {X  -140.816, Y  +291.260, Z    +0.000, E1   +53.766, E3 +325758.385}
SPL {X  -128.440, Y  +273.891, Z    +0.000, E1   +47.966, E3 +325841.473}
ENDSPLINE

SPLINE
SPL {X  -131.798, Y  +278.155, Z    +0.000, E1   +45.574, E3 +325867.100}
SPL {X  -154.181, Y  +317.936, Z    +0.000, E1   +32.662, E3 +325932.436}
SPL {X  -162.537, Y  +346.536, Z    +0.000, E1   +20.123, E3 +325931.657}
SPL {X  -164.610, Y  +359.970, Z    +0.000, E1   +13.118, E3 +325926.523}
SPL {X  -165.367, Y  +368.828, Z    +0.000, E1    +8.137, E3 +325924.976}
SPL {X  -165.621, Y  +375.422, Z    +0.000, E1    +4.067, E3 +325925.853}
SPL {X  -165.650, Y  +379.733, Z    +0.000, E1    +1.160, E3 +325924.159}
SPL {X  -165.650, Y  +383.552, Z    +0.000, E1    -1.868, E3 +325923.408}
SPL {X  -165.650, Y  +388.716, Z    +0.000, E1    -7.003, E3 +325922.813}
SPL {X  -165.650, Y  +396.644, Z    +0.000, E1   -16.434, E3 +325921.432}
SPL {X  -165.650, Y  +410.885, Z    +0.000, E1   -34.864, E3 +325916.529}
SPL {X  -165.650, Y  +448.279, Z    +0.000, E1   -53.294, E3 +325934.374}
SPL {X  -165.650, Y  +465.286, Z    +0.000, E1   -55.209, E3 +325948.226}
SPL {X  -165.650, Y  +513.874, Z    +0.000, E1   -57.683, E3 +325993.035}
ENDSPLINE

SPLINE
SPL {X  -165.650, Y  +513.412, Z    +0.000, E1   -55.245, E3 +326006.630}
SPL {X  -165.650, Y  +495.869, Z    +0.000, E1   -48.812, E3 +326017.931}
ENDSPLINE

SPLINE
SPL {X  -165.650, Y  +502.040, Z    +0.000, E1   -48.856, E3 +326028.675}
SPL {X  -165.650, Y  +507.863, Z    +0.000, E1   -49.013, E3 +326038.095}
SPL {X  -165.650, Y  +512.952, Z    +0.000, E1   -48.898, E3 +326047.872}
SPL {X  -165.650, Y  +519.321, Z    +0.000, E1   -49.041, E3 +326058.340}
SPL {X  -165.650, Y  +524.312, Z    +0.000, E1   -48.855, E3 +326068.366}
SPL {X  -165.650, Y  +530.631, Z    +0.000, E1   -48.990, E3 +326078.826}
SPL {X  -165.650, Y  +536.725, Z    +0.000, E1   -48.843, E3 +326090.576}
SPL {X  -165.650, Y  +542.959, Z    +0.000, E1   -48.923, E3 +326101.191}
SPL {X  -165.650, Y  +548.939, Z    +0.000, E1   -48.968, E3 +326111.585}
SPL {X  -165.650, Y  +553.607, Z    +0.000, E1   -48.716, E3 +326121.403}
SPL {X  -165.650, Y  +562.368, Z    +0.000, E1   -49.014, E3 +326135.464}
SPL {X  -165.650, Y  +570.317, Z    +0.000, E1   -48.893, E3 +326150.206}
SPL {X  -165.650, Y  +577.487, Z    +0.000, E1   -49.001, E3 +326162.314}
SPL {X  -165.650, Y  +581.837, Z    +0.000, E1   -48.612, E3 +326172.348}
SPL {X  -165.650, Y  +588.614, Z    +0.000, E1   -49.053, E3 +326181.865}
SPL {X  -165.650, Y  +593.784, Z    +0.000, E1   -48.711, E3 +326193.151}
SPL {X  -165.650, Y  +600.281, Z    +0.000, E1   -48.957, E3 +326203.253}
SPL {X  -165.650, Y  +606.252, Z    +0.000, E1   -48.984, E3 +326213.787}
SPL {X  -165.650, Y  +612.690, Z    +0.000, E1   -49.044, E3 +326224.816}
SPL {X  -165.650, Y  +617.274, Z    +0.000, E1   -48.670, E3 +326235.265}
SPL {X  -165.650, Y  +624.267, Z    +0.000, E1   -48.953, E3 +326246.076}
SPL {X  -165.650, Y  +630.315, Z    +0.000, E1   -49.009, E3 +326256.507}
SPL {X  -165.650, Y  +635.030, Z    +0.000, E1   -48.821, E3 +326265.992}
SPL {X  -165.650, Y  +641.084, Z    +0.000, E1   -48.892, E3 +326276.474}
SPL {X  -165.650, Y  +648.143, Z    +0.000, E1   -49.033, E3 +326288.143}
SPL {X  -165.650, Y  +655.847, Z    +0.000, E1   -48.917, E3 +326302.760}
SPL {X  -165.650, Y  +663.676, Z    +0.000, E1   -48.809, E3 +326317.198}
SPL {X  -165.650, Y  +669.580, Z    +0.000, E1   -48.844, E3 +326327.537}
SPL {X  -165.650, Y  +675.734, Z    +0.000, E1   -49.021, E3 +326337.443}
SPL {X  -165.552, Y  +681.198, Z    +0.000, E1   -48.804, E3 +326348.523}
SPL {X  -165.221, Y  +687.413, Z    +0.000, E1   -48.790, E3 +326359.695}
SPL {X  -164.785, Y  +692.407, Z    +0.000, E1   -48.653, E3 +326369.410}
SPL {X  -164.074, Y  +698.293, Z    +0.000, E1   -48.857, E3 +326378.695}
SPL {X  -163.489, Y  +702.172, Z    +0.000, E1   -48.443, E3 +326388.011}
SPL {X  -162.217, Y  +709.048, Z    +0.000, E1   -48.328, E3 +326401.151}
SPL {X  -160.800, Y  +715.289, Z    +0.000, E1   -47.964, E3 +326414.159}
SPL {X  -159.392, Y  +720.602, Z    +0.000, E1   -47.892, E3 +326424.070}
SPL {X  -157.947, Y  +725.428, Z    +0.000, E1   -47.498, E3 +326434.810}
SPL {X  -155.696, Y  +732.057, Z    +0.000, E1   -47.224, E3 +326448.286}
SPL {X  -152.475, Y  +740.240, Z    +0.000, E1   -48.059, E3 +326458.116}
SPL {X  -143.211, Y  +758.749, Z    +0.000, E1   -53.445, E3 +326459.157}
SPL {X  -130.133, Y  +777.996, Z    +0.000, E1   -46.969, E3 +326554.260}
ENDSPLINE

SPLINE
SPL {X  -153.839, Y  +736.929, Z    +0.000, E1   -32.772, E3 +326627.331}
SPL {X  -162.700, Y  +706.622, Z    +0.000, E1   -19.657, E3 +326631.624}
SPL {X  -164.822, Y  +692.043, Z    +0.000, E1   -12.043, E3 +326627.263}
SPL {X  -165.501, Y  +682.513, Z    +0.000, E1    -6.586, E3 +326625.957}
SPL {X  -165.645, Y  +676.829, Z    +0.000, E1    -2.974, E3 +326625.301}
SPL {X  -165.650, Y  +673.338, Z    +0.000, E1    -0.547, E3 +326624.470}
SPL {X  -165.650, Y  +669.008, Z    +0.000, E1    +2.993, E3 +326624.287}
SPL {X  -165.650, Y  +664.048, Z    +0.000, E1    +8.230, E3 +326623.566}
SPL {X  -165.650, Y  +658.867, Z    +0.000, E1   +14.313, E3 +326622.030}
SPL {X  -165.650, Y  +650.683, Z    +0.000, E1   +24.801, E3 +326619.466}
SPL {X  -165.650, Y  +640.858, Z    +0.000, E1   +34.904, E3 +326621.209}
SPL {X  -165.650, Y  +633.111, Z    +0.000, E1   +43.522, E3 +326618.103}
SPL {X  -165.650, Y  +586.376, Z    +0.000, E1   +59.481, E3 +326637.101}
SPL {X  -165.650, Y  +536.483, Z    +0.000, E1   +57.139, E3 +326698.869}
ENDSPLINE

SPLINE
SPL {X  -165.650, Y  +560.944, Z    +0.000, E1   +48.666, E3 +326713.891}
ENDSPLINE

SPLINE
SPL {X  -165.650, Y  +556.469, Z    +0.000, E1   +47.823, E3 +326726.830}
SPL {X  -165.650, Y  +549.545, Z    +0.000, E1   +47.953, E3 +326738.955}
SPL {X  -165.650, Y  +544.306, Z    +0.000, E1   +47.619, E3 +326750.514}
SPL {X  -165.650, Y  +537.837, Z    +0.000, E1   +47.880, E3 +326761.040}
SPL {X  -165.650, Y  +530.616, Z    +0.000, E1   +47.886, E3 +326774.405}
SPL {X  -165.650, Y  +522.460, Z    +0.000, E1   +47.738, E3 +326790.515}
SPL {X  -165.650, Y  +512.416, Z    +0.000, E1   +48.035, E3 +326807.279}
SPL {X  -165.650, Y  +507.257, Z    +0.000, E1   +47.748, E3 +326818.347}
SPL {X  -165.650, Y  +501.812, Z    +0.000, E1   +47.738, E3 +326828.630}
SPL {X  -165.650, Y  +494.522, Z    +0.000, E1   +48.055, E3 +326840.157}
SPL {X  -165.650, Y  +489.529, Z    +0.000, E1   +47.849, E3 +326850.610}
SPL {X  -165.650, Y  +484.859, Z    +0.000, E1   +47.688, E3 +326860.181}
SPL {X  -165.650, Y  +479.821, Z    +0.000, E1   +47.727, E3 +326869.349}
SPL {X  -165.650, Y  +472.739, Z    +0.000, E1   +47.923, E3 +326881.368}
SPL {X  -165.650, Y  +465.366, Z    +0.000, E1   +47.775, E3 +326895.948}
SPL {X  -165.650, Y  +457.811, Z    +0.000, E1   +47.987, E3 +326908.565}
SPL {X  -165.650, Y  +451.187, Z    +0.000, E1   +47.917, E3 +326921.308}
SPL {X  -165.650, Y  +439.019, Z    +0.000, E1   +49.830, E3 +326931.631}
SPL {X  -165.650, Y  +435.473, Z    +0.000, E1   +49.263, E3 +326941.352}
SPL {X  -165.650, Y  +428.379, Z    +0.000, E1   +49.373, E3 +326953.124}
SPL {X  -165.650, Y  +423.272, Z    +0.000, E1   +49.176, E3 +326963.259}
SPL {X  -165.650, Y  +416.522, Z    +0.000, E1   +49.338, E3 +326974.237}
SPL {X  -165.650, Y  +410.777, Z    +0.000, E1   +49.173, E3 +326985.290}
SPL {X  -165.650, Y  +402.476, Z    +0.000, E1   +49.356, E3 +326998.976}
SPL {X  -165.650, Y  +393.708, Z    +0.000, E1   +49.252, E3 +327014.966}
SPL {X  -165.650, Y  +386.526, Z    +0.000, E1   +49.193, E3 +327027.912}
SPL {X  -165.650, Y  +381.684, Z    +0.000, E1   +49.061, E3 +327037.196}
SPL {X  -165.602, Y  +374.507, Z    +0.000, E1   +49.269, E3 +327048.788}
SPL {X  -165.255, Y  +367.073, Z    +0.000, E1   +49.394, E3 +327060.981}
SPL {X  -164.828, Y  +362.023, Z    +0.000, E1   +48.964, E3 +327072.497}
SPL {X  -163.908, Y  +354.543, Z    +0.000, E1   +49.169, E3 +327084.444}
SPL {X  -163.052, Y  +349.277, Z    +0.000, E1   +48.680, E3 +327096.550}
SPL {X  -162.125, Y  +344.507, Z    +0.000, E1   +48.543, E3 +327105.690}
SPL {X  -160.947, Y  +339.310, Z    +0.000, E1   +48.561, E3 +327114.799}
SPL {X  -159.860, Y  +335.086, Z    +0.000, E1   +48.145, E3 +327124.511}
SPL {X  -158.277, Y  +329.631, Z    +0.000, E1   +47.981, E3 +327135.133}
SPL {X  -156.804, Y  +325.092, Z    +0.000, E1   +47.609, E3 +327145.026}
SPL {X  -155.465, Y  +321.311, Z    +0.000, E1   +47.446, E3 +327152.561}
SPL {X  -153.706, Y  +316.739, Z    +0.000, E1   +47.523, E3 +327160.174}
SPL {X  -143.727, Y  +296.145, Z    +0.000, E1   +53.260, E3 +327163.317}
SPL {X  -128.440, Y  +273.891, Z    +0.000, E1   +47.966, E3 +327250.564}
ENDSPLINE

SPLINE
SPL {X  -131.798, Y  +278.155, Z    +0.000, E1   +45.574, E3 +327276.191}
SPL {X  -154.181, Y  +317.936, Z    +0.000, E1   +32.662, E3 +327341.527}
SPL {X  -162.537, Y  +346.536, Z    +0.000, E1   +20.123, E3 +327340.748}
SPL {X  -165.197, Y  +366.255, Z    +0.000, E1    +9.700, E3 +327334.543}
SPL {X  -165.621, Y  +375.422, Z    +0.000, E1    +4.067, E3 +327334.943}
SPL {X  -165.650, Y  +379.733, Z    +0.000, E1    +1.160, E3 +327333.249}
SPL {X  -165.650, Y  +383.552, Z    +0.000, E1    -1.868, E3 +327332.499}
SPL {X  -165.650, Y  +388.716, Z    +0.000, E1    -7.003, E3 +327331.904}
SPL {X  -165.650, Y  +396.644, Z    +0.000, E1   -16.434, E3 +327330.523}
SPL {X  -165.650, Y  +410.885, Z    +0.000, E1   -34.864, E3 +327325.620}
SPL {X  -165.650, Y  +448.279, Z    +0.000, E1   -53.294, E3 +327343.465}
SPL {X  -165.650, Y  +465.286, Z    +0.000, E1   -55.209, E3 +327357.317}
SPL {X  -165.650, Y  +513.780, Z    +0.000, E1   -56.183, E3 +327410.833}
ENDSPLINE

SPLINE
SPL {X  -165.650, Y  +495.869, Z    +0.000, E1   -48.812, E3 +327427.022}
ENDSPLINE

SPLINE
SPL {X  -165.650, Y  +502.040, Z    +0.000, E1   -48.856, E3 +327437.766}
SPL {X  -165.650, Y  +507.863, Z    +0.000, E1   -49.013, E3 +327447.186}
SPL {X  -165.650, Y  +512.952, Z    +0.000, E1   -48.898, E3 +327456.963}
SPL {X  -165.650, Y  +519.321, Z    +0.000, E1   -49.041, E3 +327467.431}
SPL {X  -165.650, Y  +524.312, Z    +0.000, E1   -48.855, E3 +327477.457}
SPL {X  -165.650, Y  +532.191, Z    +0.000, E1   -48.944, E3 +327491.125}
SPL {X  -165.650, Y  +541.400, Z    +0.000, E1   -48.945, E3 +327507.499}
SPL {X  -165.650, Y  +548.939, Z    +0.000, E1   -48.968, E3 +327520.676}
SPL {X  -165.650, Y  +553.607, Z    +0.000, E1   -48.716, E3 +327530.494}
SPL {X  -165.650, Y  +562.368, Z    +0.000, E1   -49.014, E3 +327544.555}
SPL {X  -165.650, Y  +570.317, Z    +0.000, E1   -48.893, E3 +327559.297}
SPL {X  -165.650, Y  +577.487, Z    +0.000, E1   -49.001, E3 +327571.405}
SPL {X  -165.650, Y  +581.837, Z    +0.000, E1   -48.612, E3 +327581.439}
SPL {X  -165.650, Y  +588.614, Z    +0.000, E1   -49.053, E3 +327590.956}
SPL {X  -165.650, Y  +593.784, Z    +0.000, E1   -48.711, E3 +327602.242}
SPL {X  -165.650, Y  +600.281, Z    +0.000, E1   -48.957, E3 +327612.344}
SPL {X  -165.650, Y  +606.252, Z    +0.000, E1   -48.984, E3 +327622.878}
SPL {X  -165.650, Y  +612.690, Z    +0.000, E1   -49.044, E3 +327633.907}
SPL {X  -165.650, Y  +617.274, Z    +0.000, E1   -48.670, E3 +327644.356}
SPL {X  -165.650, Y  +624.267, Z    +0.000, E1   -48.953, E3 +327655.167}
SPL {X  -165.650, Y  +632.510, Z    +0.000, E1   -48.976, E3 +327669.922}
SPL {X  -165.650, Y  +641.084, Z    +0.000, E1   -48.892, E3 +327685.564}
SPL {X  -165.650, Y  +648.143, Z    +0.000, E1   -49.033, E3 +327697.234}
SPL {X  -165.650, Y  +655.847, Z    +0.000, E1   -48.917, E3 +327711.851}
SPL {X  -165.650, Y  +663.676, Z    +0.000, E1   -48.809, E3 +327726.289}
SPL {X  -165.650, Y  +669.580, Z    +0.000, E1   -48.844, E3 +327736.628}
SPL {X  -165.650, Y  +675.734, Z    +0.000, E1   -49.021, E3 +327746.534}
SPL {X  -165.552, Y  +681.198, Z    +0.000, E1   -48.804, E3 +327757.614}
SPL {X  -165.221, Y  +687.413, Z    +0.000, E1   -48.790, E3 +327768.786}
SPL {X  -164.785, Y  +692.407, Z    +0.000, E1   -48.653, E3 +327778.501}
SPL {X  -164.074, Y  +698.293, Z    +0.000, E1   -48.857, E3 +327787.785}
SPL {X  -163.489, Y  +702.172, Z    +0.000, E1   -48.443, E3 +327797.102}
SPL {X  -162.217, Y  +709.048, Z    +0.000, E1   -48.328, E3 +327810.242}
SPL {X  -160.800, Y  +715.289, Z    +0.000, E1   -47.964, E3 +327823.250}
SPL {X  -159.392, Y  +720.602, Z    +0.000, E1   -47.892, E3 +327833.161}
SPL {X  -157.947, Y  +725.428, Z    +0.000, E1   -47.498, E3 +327843.900}
SPL {X  -156.133, Y  +730.838, Z    +0.000, E1   -47.305, E3 +327854.617}
SPL {X  -153.862, Y  +736.871, Z    +0.000, E1   -47.425, E3 +327864.604}
SPL {X  -143.211, Y  +758.749, Z    +0.000, E1   -53.445, E3 +327868.248}
SPL {X  -130.133, Y  +777.996, Z    +0.000, E1   -46.969, E3 +327963.351}
ENDSPLINE

SPLINE
SPL {X  -153.839, Y  +736.929, Z    +0.000, E1   -32.772, E3 +328036.422}
SPL {X  -162.700, Y  +706.622, Z    +0.000, E1   -19.657, E3 +328040.715}
SPL {X  -164.822, Y  +692.043, Z    +0.000, E1   -12.043, E3 +328036.354}
SPL {X  -165.501, Y  +682.513, Z    +0.000, E1    -6.586, E3 +328035.048}
SPL {X  -165.645, Y  +676.829, Z    +0.000, E1    -2.974, E3 +328034.392}
SPL {X  -165.650, Y  +673.338, Z    +0.000, E1    -0.547, E3 +328033.561}
SPL {X  -165.650, Y  +670.475, Z    +0.000, E1    +1.794, E3 +328033.484}
SPL {X  -165.650, Y  +667.655, Z    +0.000, E1    +4.420, E3 +328033.280}
SPL {X  -165.650, Y  +664.048, Z    +0.000, E1    +8.230, E3 +328032.657}
SPL {X  -165.650, Y  +658.867, Z    +0.000, E1   +14.313, E3 +328031.121}
SPL {X  -165.650, Y  +650.683, Z    +0.000, E1   +24.801, E3 +328028.557}
SPL {X  -165.650, Y  +640.858, Z    +0.000, E1   +34.904, E3 +328030.300}
SPL {X  -165.650, Y  +633.111, Z    +0.000, E1   +43.522, E3 +328027.194}
SPL {X  -165.650, Y  +594.935, Z    +0.000, E1   +58.150, E3 +328041.794}
SPL {X  -165.650, Y  +579.579, Z    +0.000, E1   +60.394, E3 +328049.678}
SPL {X  -165.650, Y  +536.483, Z    +0.000, E1   +57.139, E3 +328107.960}
ENDSPLINE

SPLINE
SPL {X  -165.650, Y  +561.248, Z    +0.000, E1   +49.247, E3 +328118.650}
ENDSPLINE

SPLINE
SPL {X  -165.650, Y  +558.330, Z    +0.000, E1   +47.867, E3 +328132.374}
SPL {X  -165.650, Y  +550.626, Z    +0.000, E1   +48.045, E3 +328145.385}
SPL {X  -165.650, Y  +545.464, Z    +0.000, E1   +47.668, E3 +328157.253}
SPL {X  -165.650, Y  +535.912, Z    +0.000, E1   +47.888, E3 +328173.839}
SPL {X  -165.650, Y  +526.169, Z    +0.000, E1   +47.853, E3 +328192.019}
SPL {X  -165.650, Y  +517.493, Z    +0.000, E1   +47.895, E3 +328207.767}
SPL {X  -165.650, Y  +511.255, Z    +0.000, E1   +47.920, E3 +328219.056}
SPL {X  -165.650, Y  +507.257, Z    +0.000, E1   +47.748, E3 +328227.437}
SPL {X  -165.650, Y  +501.812, Z    +0.000, E1   +47.738, E3 +328237.721}
SPL {X  -165.650, Y  +494.522, Z    +0.000, E1   +48.055, E3 +328249.248}
SPL {X  -165.650, Y  +489.529, Z    +0.000, E1   +47.849, E3 +328259.701}
SPL {X  -165.650, Y  +484.859, Z    +0.000, E1   +47.688, E3 +328269.272}
SPL {X  -165.650, Y  +477.718, Z    +0.000, E1   +47.870, E3 +328281.606}
SPL {X  -165.650, Y  +469.088, Z    +0.000, E1   +47.982, E3 +328296.825}
SPL {X  -165.650, Y  +464.575, Z    +0.000, E1   +47.451, E3 +328308.240}
SPL {X  -165.650, Y  +456.851, Z    +0.000, E1   +47.856, E3 +328320.345}
SPL {X  -165.650, Y  +449.262, Z    +0.000, E1   +48.080, E3 +328332.911}
SPL {X  -165.650, Y  +436.454, Z    +0.000, E1   +49.483, E3 +328347.618}
SPL {X  -165.650, Y  +428.379, Z    +0.000, E1   +49.373, E3 +328362.214}
SPL {X  -165.650, Y  +423.272, Z    +0.000, E1   +49.176, E3 +328372.350}
SPL {X  -165.650, Y  +416.522, Z    +0.000, E1   +49.338, E3 +328383.328}
SPL {X  -165.650, Y  +410.777, Z    +0.000, E1   +49.173, E3 +328394.381}
SPL {X  -165.650, Y  +405.230, Z    +0.000, E1   +49.266, E3 +328403.584}
SPL {X  -165.650, Y  +398.850, Z    +0.000, E1   +49.279, E3 +328414.875}
SPL {X  -165.650, Y  +391.803, Z    +0.000, E1   +49.319, E3 +328426.913}
SPL {X  -165.650, Y  +386.526, Z    +0.000, E1   +49.193, E3 +328437.002}
SPL {X  -165.650, Y  +381.684, Z    +0.000, E1   +49.061, E3 +328446.287}
SPL {X  -165.602, Y  +374.507, Z    +0.000, E1   +49.269, E3 +328457.879}
SPL {X  -165.255, Y  +367.073, Z    +0.000, E1   +49.394, E3 +328470.072}
SPL {X  -164.828, Y  +362.023, Z    +0.000, E1   +48.964, E3 +328481.588}
SPL {X  -163.908, Y  +354.543, Z    +0.000, E1   +49.169, E3 +328493.535}
SPL {X  -163.052, Y  +349.277, Z    +0.000, E1   +48.680, E3 +328505.641}
SPL {X  -162.125, Y  +344.507, Z    +0.000, E1   +48.543, E3 +328514.781}
SPL {X  -160.947, Y  +339.310, Z    +0.000, E1   +48.561, E3 +328523.889}
SPL {X  -159.499, Y  +333.778, Z    +0.000, E1   +48.145, E3 +328536.002}
SPL {X  -157.957, Y  +328.606, Z    +0.000, E1   +47.890, E3 +328546.426}
SPL {X  -156.095, Y  +323.055, Z    +0.000, E1   +47.566, E3 +328558.111}
SPL {X  -153.706, Y  +316.739, Z    +0.000, E1   +47.523, E3 +328569.265}
SPL {X  -146.106, Y  +300.443, Z    +0.000, E1   +52.765, E3 +328568.884}
SPL {X  -140.816, Y  +291.260, Z    +0.000, E1   +53.766, E3 +328576.567}
SPL {X  -128.440, Y  +273.891, Z    +0.000, E1   +47.966, E3 +328659.655}
ENDSPLINE

SPLINE
SPL {X  -131.798, Y  +278.155, Z    +0.000, E1   +45.574, E3 +328685.282}
SPL {X  -154.181, Y  +317.936, Z    +0.000, E1   +32.662, E3 +328750.618}
SPL {X  -162.537, Y  +346.536, Z    +0.000, E1   +20.123, E3 +328749.838}
SPL {X  -164.610, Y  +359.970, Z    +0.000, E1   +13.118, E3 +328744.705}
SPL {X  -165.367, Y  +368.828, Z    +0.000, E1    +8.137, E3 +328743.158}
SPL {X  -165.621, Y  +375.422, Z    +0.000, E1    +4.067, E3 +328744.034}
SPL {X  -165.650, Y  +380.991, Z    +0.000, E1    +0.306, E3 +328742.046}
SPL {X  -165.650, Y  +386.066, Z    +0.000, E1    -4.211, E3 +328741.442}
SPL {X  -165.650, Y  +392.013, Z    +0.000, E1   -10.856, E3 +328740.424}
SPL {X  -165.650, Y  +398.769, Z    +0.000, E1   -19.304, E3 +328739.035}
SPL {X  -165.650, Y  +407.471, Z    +0.000, E1   -31.017, E3 +328735.194}
SPL {X  -165.650, Y  +414.706, Z    +0.000, E1   -39.242, E3 +328734.170}
SPL {X  -165.650, Y  +448.279, Z    +0.000, E1   -53.294, E3 +328752.556}
SPL {X  -165.650, Y  +465.286, Z    +0.000, E1   -55.209, E3 +328766.408}
SPL {X  -165.650, Y  +513.780, Z    +0.000, E1   -56.183, E3 +328819.924}
ENDSPLINE

SPLINE
SPL {X  -165.650, Y  +495.869, Z    +0.000, E1   -48.812, E3 +328836.113}
ENDSPLINE

SPLINE
SPL {X  -165.650, Y  +502.040, Z    +0.000, E1   -48.856, E3 +328846.857}
SPL {X  -165.650, Y  +507.863, Z    +0.000, E1   -49.013, E3 +328856.277}
SPL {X  -165.650, Y  +512.952, Z    +0.000, E1   -48.898, E3 +328866.054}
SPL {X  -165.650, Y  +519.321, Z    +0.000, E1   -49.041, E3 +328876.522}
SPL {X  -165.650, Y  +524.312, Z    +0.000, E1   -48.855, E3 +328886.548}
SPL {X  -165.650, Y  +532.191, Z    +0.000, E1   -48.944, E3 +328900.216}
SPL {X  -165.650, Y  +541.400, Z    +0.000, E1   -48.945, E3 +328916.590}
SPL {X  -165.650, Y  +548.939, Z    +0.000, E1   -48.968, E3 +328929.767}
SPL {X  -165.650, Y  +553.607, Z    +0.000, E1   -48.716, E3 +328939.585}
SPL {X  -165.650, Y  +562.368, Z    +0.000, E1   -49.014, E3 +328953.645}
SPL {X  -165.650, Y  +570.317, Z    +0.000, E1   -48.893, E3 +328968.388}
SPL {X  -165.650, Y  +577.487, Z    +0.000, E1   -49.001, E3 +328980.496}
SPL {X  -165.650, Y  +581.837, Z    +0.000, E1   -48.612, E3 +328990.530}
SPL {X  -165.650, Y  +588.614, Z    +0.000, E1   -49.053, E3 +329000.047}
SPL {X  -165.650, Y  +593.784, Z    +0.000, E1   -48.711, E3 +329011.333}
SPL {X  -165.650, Y  +600.281, Z    +0.000, E1   -48.957, E3 +329021.435}
SPL {X  -165.650, Y  +606.252, Z    +0.000, E1   -48.984, E3 +329031.969}
SPL {X  -165.650, Y  +612.690, Z    +0.000, E1   -49.044, E3 +329042.997}
SPL {X  -165.650, Y  +617.274, Z    +0.000, E1   -48.670, E3 +329053.447}
SPL {X  -165.650, Y  +624.267, Z    +0.000, E1   -48.953, E3 +329064.258}
SPL {X  -165.650, Y  +632.510, Z    +0.000, E1   -48.976, E3 +329079.013}
SPL {X  -165.650, Y  +641.084, Z    +0.000, E1   -48.892, E3 +329094.655}
SPL {X  -165.650, Y  +648.143, Z    +0.000, E1   -49.033, E3 +329106.324}
SPL {X  -165.650, Y  +655.847, Z    +0.000, E1   -48.917, E3 +329120.942}
SPL {X  -165.650, Y  +663.676, Z    +0.000, E1   -48.809, E3 +329135.380}
SPL {X  -165.650, Y  +669.580, Z    +0.000, E1   -48.844, E3 +329145.719}
SPL {X  -165.650, Y  +675.734, Z    +0.000, E1   -49.021, E3 +329155.625}
SPL {X  -165.552, Y  +681.198, Z    +0.000, E1   -48.804, E3 +329166.705}
SPL {X  -165.221, Y  +687.413, Z    +0.000, E1   -48.790, E3 +329177.877}
SPL {X  -164.785, Y  +692.407, Z    +0.000, E1   -48.653, E3 +329187.592}
SPL {X  -164.074, Y  +698.293, Z    +0.000, E1   -48.857, E3 +329196.876}
SPL {X  -163.489, Y  +702.172, Z    +0.000, E1   -48.443, E3 +329206.193}
SPL {X  -162.217, Y  +709.048, Z    +0.000, E1   -48.328, E3 +329219.333}
SPL {X  -160.800, Y  +715.289, Z    +0.000, E1   -47.964, E3 +329232.341}
SPL {X  -159.392, Y  +720.602, Z    +0.000, E1   -47.892, E3 +329242.252}
SPL {X  -157.947, Y  +725.428, Z    +0.000, E1   -47.498, E3 +329252.991}
SPL {X  -156.133, Y  +730.838, Z    +0.000, E1   -47.305, E3 +329263.708}
SPL {X  -153.862, Y  +736.871, Z    +0.000, E1   -47.425, E3 +329273.695}
SPL {X  -143.211, Y  +758.749, Z    +0.000, E1   -53.445, E3 +329277.339}
SPL {X  -129.526, Y  +778.761, Z    +0.000, E1   -47.396, E3 +329368.080}
ENDSPLINE

SPLINE
SPL {X  -152.848, Y  +739.355, Z    +0.000, E1   -33.672, E3 +329443.649}
SPL {X  -162.700, Y  +706.622, Z    +0.000, E1   -19.657, E3 +329449.806}
SPL {X  -164.822, Y  +692.043, Z    +0.000, E1   -12.043, E3 +329445.445}
SPL {X  -165.501, Y  +682.513, Z    +0.000, E1    -6.586, E3 +329444.139}
SPL {X  -165.645, Y  +676.829, Z    +0.000, E1    -2.974, E3 +329443.483}
SPL {X  -165.650, Y  +673.338, Z    +0.000, E1    -0.547, E3 +329442.652}
SPL {X  -165.650, Y  +670.475, Z    +0.000, E1    +1.794, E3 +329442.575}
SPL {X  -165.650, Y  +667.655, Z    +0.000, E1    +4.420, E3 +329442.371}
SPL {X  -165.650, Y  +664.048, Z    +0.000, E1    +8.230, E3 +329441.748}
SPL {X  -165.650, Y  +658.867, Z    +0.000, E1   +14.313, E3 +329440.212}
SPL {X  -165.650, Y  +650.683, Z    +0.000, E1   +24.801, E3 +329437.647}
SPL {X  -165.650, Y  +636.402, Z    +0.000, E1   +39.824, E3 +329437.610}
SPL {X  -165.650, Y  +594.935, Z    +0.000, E1   +58.150, E3 +329450.885}
SPL {X  -165.650, Y  +579.579, Z    +0.000, E1   +60.394, E3 +329458.769}
SPL {X  -165.650, Y  +536.483, Z    +0.000, E1   +57.139, E3 +329517.051}
ENDSPLINE

SPLINE
SPL {X  -165.650, Y  +561.248, Z    +0.000, E1   +49.247, E3 +329527.741}
ENDSPLINE

SPLINE
SPL {X  -165.650, Y  +558.330, Z    +0.000, E1   +47.867, E3 +329541.465}
SPL {X  -165.650, Y  +550.626, Z    +0.000, E1   +48.045, E3 +329554.475}
SPL {X  -165.650, Y  +545.464, Z    +0.000, E1   +47.668, E3 +329566.344}
SPL {X  -165.650, Y  +537.837, Z    +0.000, E1   +47.880, E3 +329579.221}
SPL {X  -165.650, Y  +530.616, Z    +0.000, E1   +47.886, E3 +329592.587}
SPL {X  -165.650, Y  +522.460, Z    +0.000, E1   +47.738, E3 +329608.697}
SPL {X  -165.650, Y  +512.416, Z    +0.000, E1   +48.035, E3 +329625.461}
SPL {X  -165.650, Y  +507.257, Z    +0.000, E1   +47.748, E3 +329636.528}
SPL {X  -165.650, Y  +501.812, Z    +0.000, E1   +47.738, E3 +329646.812}
SPL {X  -165.650, Y  +493.465, Z    +0.000, E1   +47.959, E3 +329660.982}
SPL {X  -165.650, Y  +486.149, Z    +0.000, E1   +47.831, E3 +329675.257}
SPL {X  -165.650, Y  +479.821, Z    +0.000, E1   +47.727, E3 +329687.531}
SPL {X  -165.650, Y  +472.739, Z    +0.000, E1   +47.923, E3 +329699.550}
SPL {X  -165.650, Y  +465.366, Z    +0.000, E1   +47.775, E3 +329714.130}
SPL {X  -165.650, Y  +456.851, Z    +0.000, E1   +47.856, E3 +329729.436}
SPL {X  -165.650, Y  +449.262, Z    +0.000, E1   +48.080, E3 +329742.002}
SPL {X  -165.650, Y  +436.454, Z    +0.000, E1   +49.483, E3 +329756.709}
SPL {X  -165.650, Y  +428.379, Z    +0.000, E1   +49.373, E3 +329771.305}
SPL {X  -165.650, Y  +421.000, Z    +0.000, E1   +49.266, E3 +329785.053}
SPL {X  -165.650, Y  +412.094, Z    +0.000, E1   +49.264, E3 +329800.740}
SPL {X  -165.650, Y  +405.230, Z    +0.000, E1   +49.266, E3 +329812.675}
SPL {X  -165.650, Y  +400.266, Z    +0.000, E1   +49.362, E3 +329820.841}
SPL {X  -165.650, Y  +393.708, Z    +0.000, E1   +49.252, E3 +329833.148}
SPL {X  -165.650, Y  +386.526, Z    +0.000, E1   +49.193, E3 +329846.093}
SPL {X  -165.649, Y  +378.059, Z    +0.000, E1   +49.283, E3 +329860.636}
SPL {X  -165.292, Y  +367.617, Z    +0.000, E1   +49.239, E3 +329879.401}
SPL {X  -164.692, Y  +360.715, Z    +0.000, E1   +48.960, E3 +329892.935}
SPL {X  -163.908, Y  +354.543, Z    +0.000, E1   +49.169, E3 +329902.626}
SPL {X  -163.052, Y  +349.277, Z    +0.000, E1   +48.680, E3 +329914.732}
SPL {X  -162.125, Y  +344.507, Z    +0.000, E1   +48.543, E3 +329923.871}
SPL {X  -160.947, Y  +339.310, Z    +0.000, E1   +48.561, E3 +329932.980}
SPL {X  -159.499, Y  +333.778, Z    +0.000, E1   +48.145, E3 +329945.093}
SPL {X  -157.380, Y  +326.814, Z    +0.000, E1   +47.797, E3 +329959.364}
SPL {X  -155.465, Y  +321.311, Z    +0.000, E1   +47.446, E3 +329970.742}
SPL {X  -153.706, Y  +316.739, Z    +0.000, E1   +47.523, E3 +329978.356}
SPL {X  -143.727, Y  +296.145, Z    +0.000, E1   +53.260, E3 +329981.499}
SPL {X  -128.440, Y  +273.891, Z    +0.000, E1   +47.966, E3 +330068.745}
ENDSPLINE

SPLINE
SPL {X  -131.798, Y  +278.155, Z    +0.000, E1   +45.574, E3 +330094.372}
SPL {X  -154.181, Y  +317.936, Z    +0.000, E1   +32.662, E3 +330159.709}
SPL {X  -162.537, Y  +346.536, Z    +0.000, E1   +20.123, E3 +330158.929}
SPL {X  -164.610, Y  +359.970, Z    +0.000, E1   +13.118, E3 +330153.796}
SPL {X  -165.367, Y  +368.828, Z    +0.000, E1    +8.137, E3 +330152.248}
SPL {X  -165.621, Y  +375.422, Z    +0.000, E1    +4.067, E3 +330153.125}
SPL {X  -165.650, Y  +380.991, Z    +0.000, E1    +0.306, E3 +330151.137}
SPL {X  -165.650, Y  +386.066, Z    +0.000, E1    -4.211, E3 +330150.533}
SPL {X  -165.650, Y  +392.013, Z    +0.000, E1   -10.856, E3 +330149.515}
SPL {X  -165.650, Y  +398.769, Z    +0.000, E1   -19.304, E3 +330148.126}
SPL {X  -165.650, Y  +410.885, Z    +0.000, E1   -34.864, E3 +330143.802}
SPL {X  -165.650, Y  +446.037, Z    +0.000, E1   -53.739, E3 +330157.866}
SPL {X  -165.650, Y  +454.158, Z    +0.000, E1   -53.343, E3 +330168.218}
SPL {X  -165.650, Y  +513.780, Z    +0.000, E1   -56.183, E3 +330229.015}
ENDSPLINE

SPLINE
SPL {X  -165.650, Y  +495.869, Z    +0.000, E1   -48.812, E3 +330245.204}
ENDSPLINE

SPLINE
SPL {X  -165.650, Y  +502.040, Z    +0.000, E1   -48.856, E3 +330255.948}
SPL {X  -165.650, Y  +507.863, Z    +0.000, E1   -49.013, E3 +330265.368}
SPL {X  -165.650, Y  +512.952, Z    +0.000, E1   -48.898, E3 +330275.145}
SPL {X  -165.650, Y  +519.321, Z    +0.000, E1   -49.041, E3 +330285.613}
SPL {X  -165.650, Y  +524.312, Z    +0.000, E1   -48.855, E3 +330295.638}
SPL {X  -165.650, Y  +532.191, Z    +0.000, E1   -48.944, E3 +330309.307}
SPL {X  -165.650, Y  +541.400, Z    +0.000, E1   -48.945, E3 +330325.681}
SPL {X  -165.650, Y  +548.939, Z    +0.000, E1   -48.968, E3 +330338.858}
SPL {X  -165.650, Y  +553.607, Z    +0.000, E1   -48.716, E3 +330348.676}
SPL {X  -165.650, Y  +562.368, Z    +0.000, E1   -49.014, E3 +330362.736}
SPL {X  -165.650, Y  +570.317, Z    +0.000, E1   -48.893, E3 +330377.479}
SPL {X  -165.650, Y  +577.487, Z    +0.000, E1   -49.001, E3 +330389.587}
SPL {X  -165.650, Y  +581.837, Z    +0.000, E1   -48.612, E3 +330399.621}
SPL {X  -165.650, Y  +588.614, Z    +0.000, E1   -49.053, E3 +330409.138}
SPL {X  -165.650, Y  +593.784, Z    +0.000, E1   -48.711, E3 +330420.424}
SPL {X  -165.650, Y  +600.281, Z    +0.000, E1   -48.957, E3 +330430.526}
SPL {X  -165.650, Y  +606.252, Z    +0.000, E1   -48.984, E3 +330441.060}
SPL {X  -165.650, Y  +612.690, Z    +0.000, E1   -49.044, E3 +330452.088}
SPL {X  -165.650, Y  +617.274, Z    +0.000, E1   -48.670, E3 +330462.537}
SPL {X  -165.650, Y  +624.267, Z    +0.000, E1   -48.953, E3 +330473.349}
SPL {X  -165.650, Y  +632.510, Z    +0.000, E1   -48.976, E3 +330488.104}
SPL {X  -165.650, Y  +641.084, Z    +0.000, E1   -48.892, E3 +330503.746}
SPL {X  -165.650, Y  +648.143, Z    +0.000, E1   -49.033, E3 +330515.415}
SPL {X  -165.650, Y  +655.847, Z    +0.000, E1   -48.917, E3 +330530.033}
SPL {X  -165.650, Y  +663.676, Z    +0.000, E1   -48.809, E3 +330544.471}
SPL {X  -165.650, Y  +669.580, Z    +0.000, E1   -48.844, E3 +330554.810}
SPL {X  -165.650, Y  +675.734, Z    +0.000, E1   -49.021, E3 +330564.716}
SPL {X  -165.552, Y  +681.198, Z    +0.000, E1   -48.804, E3 +330575.796}
SPL {X  -165.221, Y  +687.413, Z    +0.000, E1   -48.790, E3 +330586.968}
SPL {X  -164.785, Y  +692.407, Z    +0.000, E1   -48.653, E3 +330596.683}
SPL {X  -164.074, Y  +698.293, Z    +0.000, E1   -48.857, E3 +330605.967}
SPL {X  -163.489, Y  +702.172, Z    +0.000, E1   -48.443, E3 +330615.284}
SPL {X  -162.217, Y  +709.048, Z    +0.000, E1   -48.328, E3 +330628.424}
SPL {X  -160.800, Y  +715.289, Z    +0.000, E1   -47.964, E3 +330641.432}
SPL {X  -159.392, Y  +720.602, Z    +0.000, E1   -47.892, E3 +330651.343}
SPL {X  -157.947, Y  +725.428, Z    +0.000, E1   -47.498, E3 +330662.082}
SPL {X  -156.133, Y  +730.838, Z    +0.000, E1   -47.305, E3 +330672.799}
SPL {X  -153.862, Y  +736.871, Z    +0.000, E1   -47.425, E3 +330682.786}
SPL {X  -143.211, Y  +758.749, Z    +0.000, E1   -53.445, E3 +330686.429}
SPL {X  -129.526, Y  +778.761, Z    +0.000, E1   -47.396, E3 +330777.171}
ENDSPLINE

SPLINE
SPL {X  -152.848, Y  +739.355, Z    +0.000, E1   -33.672, E3 +330852.740}
SPL {X  -162.700, Y  +706.622, Z    +0.000, E1   -19.657, E3 +330858.897}
SPL {X  -164.822, Y  +692.043, Z    +0.000, E1   -12.043, E3 +330854.536}
SPL {X  -165.501, Y  +682.513, Z    +0.000, E1    -6.586, E3 +330853.230}
SPL {X  -165.645, Y  +676.829, Z    +0.000, E1    -2.974, E3 +330852.573}
SPL {X  -165.650, Y  +673.338, Z    +0.000, E1    -0.547, E3 +330851.743}
SPL {X  -165.650, Y  +670.475, Z    +0.000, E1    +1.794, E3 +330851.666}
SPL {X  -165.650, Y  +667.655, Z    +0.000, E1    +4.420, E3 +330851.462}
SPL {X  -165.650, Y  +664.048, Z    +0.000, E1    +8.230, E3 +330850.839}
SPL {X  -165.650, Y  +658.867, Z    +0.000, E1   +14.313, E3 +330849.303}
SPL {X  -165.650, Y  +650.683, Z    +0.000, E1   +24.801, E3 +330846.738}
SPL {X  -165.650, Y  +636.402, Z    +0.000, E1   +39.824, E3 +330846.701}
SPL {X  -165.650, Y  +594.935, Z    +0.000, E1   +58.150, E3 +330859.976}
SPL {X  -165.650, Y  +579.579, Z    +0.000, E1   +60.394, E3 +330867.860}
SPL {X  -165.650, Y  +536.483, Z    +0.000, E1   +57.139, E3 +330926.142}
ENDSPLINE

SPLINE
SPL {X  -165.650, Y  +561.248, Z    +0.000, E1   +49.247, E3 +330936.832}
ENDSPLINE

SPLINE
SPL {X  -165.650, Y  +558.330, Z    +0.000, E1   +47.867, E3 +330950.556}
SPL {X  -165.650, Y  +550.626, Z    +0.000, E1   +48.045, E3 +330963.566}
SPL {X  -165.650, Y  +545.464, Z    +0.000, E1   +47.668, E3 +330975.435}
SPL {X  -165.650, Y  +537.837, Z    +0.000, E1   +47.880, E3 +330988.312}
SPL {X  -165.650, Y  +530.616, Z    +0.000, E1   +47.886, E3 +331001.678}
SPL {X  -165.650, Y  +522.460, Z    +0.000, E1   +47.738, E3 +331017.787}
SPL {X  -165.650, Y  +512.416, Z    +0.000, E1   +48.035, E3 +331034.552}
SPL {X  -165.650, Y  +507.257, Z    +0.000, E1   +47.748, E3 +331045.619}
SPL {X  -165.650, Y  +501.812, Z    +0.000, E1   +47.738, E3 +331055.903}
SPL {X  -165.650, Y  +493.465, Z    +0.000, E1   +47.959, E3 +331070.073}
SPL {X  -165.650, Y  +486.149, Z    +0.000, E1   +47.831, E3 +331084.348}
SPL {X  -165.650, Y  +479.821, Z    +0.000, E1   +47.727, E3 +331096.622}
SPL {X  -165.650, Y  +472.739, Z    +0.000, E1   +47.923, E3 +331108.641}
SPL {X  -165.650, Y  +466.586, Z    +0.000, E1   +48.125, E3 +331118.656}
SPL {X  -165.650, Y  +464.575, Z    +0.000, E1   +47.451, E3 +331126.421}
SPL {X  -165.650, Y  +456.851, Z    +0.000, E1   +47.856, E3 +331138.527}
SPL {X  -165.650, Y  +445.317, Z    +0.000, E1   +48.773, E3 +331154.105}
SPL {X  -165.650, Y  +435.473, Z    +0.000, E1   +49.263, E3 +331168.625}
SPL {X  -165.650, Y  +428.379, Z    +0.000, E1   +49.373, E3 +331180.396}
SPL {X  -165.650, Y  +423.272, Z    +0.000, E1   +49.176, E3 +331190.532}
SPL {X  -165.650, Y  +416.522, Z    +0.000, E1   +49.338, E3 +331201.510}
SPL {X  -165.650, Y  +408.142, Z    +0.000, E1   +49.261, E3 +331216.871}
SPL {X  -165.650, Y  +400.266, Z    +0.000, E1   +49.362, E3 +331229.932}
SPL {X  -165.650, Y  +393.708, Z    +0.000, E1   +49.252, E3 +331242.239}
SPL {X  -165.650, Y  +384.475, Z    +0.000, E1   +49.187, E3 +331259.037}
SPL {X  -165.602, Y  +374.507, Z    +0.000, E1   +49.269, E3 +331276.061}
SPL {X  -165.255, Y  +367.073, Z    +0.000, E1   +49.394, E3 +331288.254}
SPL {X  -164.828, Y  +362.023, Z    +0.000, E1   +48.964, E3 +331299.769}
SPL {X  -163.908, Y  +354.543, Z    +0.000, E1   +49.169, E3 +331311.717}
SPL {X  -163.052, Y  +349.277, Z    +0.000, E1   +48.680, E3 +331323.823}
SPL {X  -162.125, Y  +344.507, Z    +0.000, E1   +48.543, E3 +331332.962}
SPL {X  -160.947, Y  +339.310, Z    +0.000, E1   +48.561, E3 +331342.071}
SPL {X  -159.860, Y  +335.086, Z    +0.000, E1   +48.145, E3 +331351.783}
SPL {X  -158.277, Y  +329.631, Z    +0.000, E1   +47.981, E3 +331362.406}
SPL {X  -156.804, Y  +325.092, Z    +0.000, E1   +47.609, E3 +331372.299}
SPL {X  -155.465, Y  +321.311, Z    +0.000, E1   +47.446, E3 +331379.833}
SPL {X  -153.706, Y  +316.739, Z    +0.000, E1   +47.523, E3 +331387.446}
SPL {X  -143.727, Y  +296.145, Z    +0.000, E1   +53.260, E3 +331390.590}
SPL {X  -128.440, Y  +273.891, Z    +0.000, E1   +47.966, E3 +331477.836}
ENDSPLINE

SPLINE
SPL {X  -131.798, Y  +278.155, Z    +0.000, E1   +45.574, E3 +331503.463}
SPL {X  -154.181, Y  +317.936, Z    +0.000, E1   +32.662, E3 +331568.800}
SPL {X  -162.537, Y  +346.536, Z    +0.000, E1   +20.123, E3 +331568.020}
SPL {X  -165.197, Y  +366.255, Z    +0.000, E1    +9.700, E3 +331561.815}
SPL {X  -165.621, Y  +375.422, Z    +0.000, E1    +4.067, E3 +331562.216}
SPL {X  -165.650, Y  +380.991, Z    +0.000, E1    +0.306, E3 +331560.228}
SPL {X  -165.650, Y  +386.066, Z    +0.000, E1    -4.211, E3 +331559.624}
SPL {X  -165.650, Y  +392.013, Z    +0.000, E1   -10.856, E3 +331558.606}
SPL {X  -165.650, Y  +398.769, Z    +0.000, E1   -19.304, E3 +331557.217}
SPL {X  -165.650, Y  +410.885, Z    +0.000, E1   -34.864, E3 +331552.893}
SPL {X  -165.650, Y  +448.279, Z    +0.000, E1   -53.294, E3 +331570.738}
SPL {X  -165.650, Y  +465.286, Z    +0.000, E1   -55.209, E3 +331584.589}
SPL {X  -165.650, Y  +513.874, Z    +0.000, E1   -57.683, E3 +331629.398}
ENDSPLINE

SPLINE
SPL {X  -165.650, Y  +513.412, Z    +0.000, E1   -55.245, E3 +331642.994}
SPL {X  -165.650, Y  +495.869, Z    +0.000, E1   -48.812, E3 +331654.295}
ENDSPLINE

SPLINE
SPL {X  -165.650, Y  +502.040, Z    +0.000, E1   -48.856, E3 +331665.039}
SPL {X  -165.650, Y  +507.863, Z    +0.000, E1   -49.013, E3 +331674.459}
SPL {X  -165.650, Y  +512.952, Z    +0.000, E1   -48.898, E3 +331684.236}
SPL {X  -165.650, Y  +519.321, Z    +0.000, E1   -49.041, E3 +331694.704}
SPL {X  -165.650, Y  +524.312, Z    +0.000, E1   -48.855, E3 +331704.729}
SPL {X  -165.650, Y  +530.631, Z    +0.000, E1   -48.990, E3 +331715.189}
SPL {X  -165.650, Y  +536.725, Z    +0.000, E1   -48.843, E3 +331726.940}
SPL {X  -165.650, Y  +542.959, Z    +0.000, E1   -48.923, E3 +331737.555}
SPL {X  -165.650, Y  +548.939, Z    +0.000, E1   -48.968, E3 +331747.949}
SPL {X  -165.650, Y  +553.607, Z    +0.000, E1   -48.716, E3 +331757.767}
SPL {X  -165.650, Y  +562.368, Z    +0.000, E1   -49.014, E3 +331771.827}
SPL {X  -165.650, Y  +570.317, Z    +0.000, E1   -48.893, E3 +331786.570}
SPL {X  -165.650, Y  +577.487, Z    +0.000, E1   -49.001, E3 +331798.678}
SPL {X  -165.650, Y  +581.837, Z    +0.000, E1   -48.612, E3 +331808.712}
SPL {X  -165.650, Y  +588.614, Z    +0.000, E1   -49.053, E3 +331818.229}
SPL {X  -165.650, Y  +593.784, Z    +0.000, E1   -48.711, E3 +331829.515}
SPL {X  -165.650, Y  +600.281, Z    +0.000, E1   -48.957, E3 +331839.617}
SPL {X  -165.650, Y  +606.252, Z    +0.000, E1   -48.984, E3 +331850.150}
SPL {X  -165.650, Y  +612.690, Z    +0.000, E1   -49.044, E3 +331861.179}
SPL {X  -165.650, Y  +617.274, Z    +0.000, E1   -48.670, E3 +331871.628}
SPL {X  -165.650, Y  +624.267, Z    +0.000, E1   -48.953, E3 +331882.440}
SPL {X  -165.650, Y  +630.315, Z    +0.000, E1   -49.009, E3 +331892.871}
SPL {X  -165.650, Y  +635.030, Z    +0.000, E1   -48.821, E3 +331902.355}
SPL {X  -165.650, Y  +641.084, Z    +0.000, E1   -48.892, E3 +331912.837}
SPL {X  -165.650, Y  +648.143, Z    +0.000, E1   -49.033, E3 +331924.506}
SPL {X  -165.650, Y  +655.847, Z    +0.000, E1   -48.917, E3 +331939.124}
SPL {X  -165.650, Y  +663.676, Z    +0.000, E1   -48.809, E3 +331953.562}
SPL {X  -165.650, Y  +669.580, Z    +0.000, E1   -48.844, E3 +331963.901}
SPL {X  -165.650, Y  +675.734, Z    +0.000, E1   -49.021, E3 +331973.807}
SPL {X  -165.552, Y  +681.198, Z    +0.000, E1   -48.804, E3 +331984.887}
SPL {X  -165.221, Y  +687.413, Z    +0.000, E1   -48.790, E3 +331996.059}
SPL {X  -164.785, Y  +692.407, Z    +0.000, E1   -48.653, E3 +332005.774}
SPL {X  -164.074, Y  +698.293, Z    +0.000, E1   -48.857, E3 +332015.058}
SPL {X  -163.489, Y  +702.172, Z    +0.000, E1   -48.443, E3 +332024.375}
SPL {X  -162.671, Y  +706.776, Z    +0.000, E1   -48.273, E3 +332033.594}
SPL {X  -161.177, Y  +713.734, Z    +0.000, E1   -48.156, E3 +332046.880}
SPL {X  -159.392, Y  +720.602, Z    +0.000, E1   -47.892, E3 +332060.434}
SPL {X  -157.947, Y  +725.428, Z    +0.000, E1   -47.498, E3 +332071.173}
SPL {X  -155.696, Y  +732.057, Z    +0.000, E1   -47.224, E3 +332084.650}
SPL {X  -152.475, Y  +740.240, Z    +0.000, E1   -48.059, E3 +332094.479}
SPL {X  -143.211, Y  +758.749, Z    +0.000, E1   -53.445, E3 +332095.520}
SPL {X  -130.133, Y  +777.996, Z    +0.000, E1   -46.969, E3 +332190.624}
ENDSPLINE

SPLINE
SPL {X  -153.839, Y  +736.929, Z    +0.000, E1   -32.772, E3 +332263.695}
SPL {X  -162.700, Y  +706.622, Z    +0.000, E1   -19.657, E3 +332267.988}
SPL {X  -164.822, Y  +692.043, Z    +0.000, E1   -12.043, E3 +332263.626}
SPL {X  -165.501, Y  +682.513, Z    +0.000, E1    -6.586, E3 +332262.321}
SPL {X  -165.645, Y  +676.829, Z    +0.000, E1    -2.974, E3 +332261.664}
SPL {X  -165.650, Y  +673.338, Z    +0.000, E1    -0.547, E3 +332260.833}
SPL {X  -165.650, Y  +669.008, Z    +0.000, E1    +2.993, E3 +332260.651}
SPL {X  -165.650, Y  +663.208, Z    +0.000, E1    +9.118, E3 +332259.735}
SPL {X  -165.650, Y  +657.399, Z    +0.000, E1   +16.251, E3 +332257.855}
SPL {X  -165.650, Y  +650.683, Z    +0.000, E1   +24.801, E3 +332255.829}
SPL {X  -165.650, Y  +636.402, Z    +0.000, E1   +39.824, E3 +332255.792}
SPL {X  -165.650, Y  +586.376, Z    +0.000, E1   +59.481, E3 +332273.464}
SPL {X  -165.650, Y  +554.310, Z    +0.000, E1   +51.914, E3 +332341.509}
ENDSPLINE

SPLINE
SPL {X  -165.650, Y  +561.648, Z    +0.000, E1   +48.058, E3 +332352.325}
ENDSPLINE

SPLINE
SPL {X  -165.650, Y  +556.469, Z    +0.000, E1   +47.823, E3 +332363.194}
SPL {X  -165.650, Y  +549.545, Z    +0.000, E1   +47.953, E3 +332375.319}
SPL {X  -165.650, Y  +541.974, Z    +0.000, E1   +47.882, E3 +332389.709}
SPL {X  -165.650, Y  +535.023, Z    +0.000, E1   +47.697, E3 +332403.697}
SPL {X  -165.650, Y  +526.169, Z    +0.000, E1   +47.853, E3 +332419.292}
SPL {X  -165.650, Y  +520.016, Z    +0.000, E1   +47.658, E3 +332431.676}
SPL {X  -165.650, Y  +512.416, Z    +0.000, E1   +48.035, E3 +332443.643}
SPL {X  -165.650, Y  +507.257, Z    +0.000, E1   +47.748, E3 +332454.710}
SPL {X  -165.650, Y  +501.812, Z    +0.000, E1   +47.738, E3 +332464.994}
SPL {X  -165.650, Y  +494.522, Z    +0.000, E1   +48.055, E3 +332476.521}
SPL {X  -165.650, Y  +489.529, Z    +0.000, E1   +47.849, E3 +332486.974}
SPL {X  -165.650, Y  +481.894, Z    +0.000, E1   +47.756, E3 +332501.875}
SPL {X  -165.650, Y  +472.739, Z    +0.000, E1   +47.923, E3 +332517.732}
SPL {X  -165.650, Y  +465.366, Z    +0.000, E1   +47.775, E3 +332532.312}
SPL {X  -165.650, Y  +457.811, Z    +0.000, E1   +47.987, E3 +332544.929}
SPL {X  -165.650, Y  +451.187, Z    +0.000, E1   +47.917, E3 +332557.672}
SPL {X  -165.650, Y  +436.765, Z    +0.000, E1   +49.819, E3 +332572.083}
SPL {X  -165.650, Y  +430.891, Z    +0.000, E1   +49.130, E3 +332586.585}
SPL {X  -165.650, Y  +423.272, Z    +0.000, E1   +49.176, E3 +332599.623}
SPL {X  -165.650, Y  +416.522, Z    +0.000, E1   +49.338, E3 +332610.601}
SPL {X  -165.650, Y  +408.142, Z    +0.000, E1   +49.261, E3 +332625.962}
SPL {X  -165.650, Y  +400.266, Z    +0.000, E1   +49.362, E3 +332639.023}
SPL {X  -165.650, Y  +393.708, Z    +0.000, E1   +49.252, E3 +332651.330}
SPL {X  -165.650, Y  +384.475, Z    +0.000, E1   +49.187, E3 +332668.128}
SPL {X  -165.602, Y  +374.507, Z    +0.000, E1   +49.269, E3 +332685.152}
SPL {X  -165.183, Y  +366.070, Z    +0.000, E1   +49.261, E3 +332700.036}
SPL {X  -164.442, Y  +358.533, Z    +0.000, E1   +49.061, E3 +332714.485}
SPL {X  -163.224, Y  +350.255, Z    +0.000, E1   +48.882, E3 +332730.205}
SPL {X  -162.125, Y  +344.507, Z    +0.000, E1   +48.543, E3 +332742.053}
SPL {X  -160.947, Y  +339.310, Z    +0.000, E1   +48.561, E3 +332751.162}
SPL {X  -159.860, Y  +335.086, Z    +0.000, E1   +48.145, E3 +332760.874}
SPL {X  -158.277, Y  +329.631, Z    +0.000, E1   +47.981, E3 +332771.497}
SPL {X  -156.095, Y  +323.055, Z    +0.000, E1   +47.566, E3 +332785.383}
SPL {X  -153.706, Y  +316.739, Z    +0.000, E1   +47.523, E3 +332796.537}
SPL {X  -146.106, Y  +300.443, Z    +0.000, E1   +52.765, E3 +332796.157}
SPL {X  -140.816, Y  +291.260, Z    +0.000, E1   +53.766, E3 +332803.840}
SPL {X  -128.440, Y  +273.891, Z    +0.000, E1   +47.966, E3 +332886.927}
ENDSPLINE

SPLINE
SPL {X  -131.798, Y  +278.155, Z    +0.000, E1   +45.574, E3 +332912.554}
SPL {X  -154.181, Y  +317.936, Z    +0.000, E1   +32.662, E3 +332977.891}
SPL {X  -162.537, Y  +346.536, Z    +0.000, E1   +20.123, E3 +332977.111}
SPL {X  -164.610, Y  +359.970, Z    +0.000, E1   +13.118, E3 +332971.977}
SPL {X  -165.367, Y  +368.828, Z    +0.000, E1    +8.137, E3 +332970.430}
SPL {X  -165.621, Y  +375.422, Z    +0.000, E1    +4.067, E3 +332971.307}
SPL {X  -165.650, Y  +379.733, Z    +0.000, E1    +1.160, E3 +332969.613}
SPL {X  -165.650, Y  +383.552, Z    +0.000, E1    -1.868, E3 +332968.863}
SPL {X  -165.650, Y  +388.716, Z    +0.000, E1    -7.003, E3 +332968.267}
SPL {X  -165.650, Y  +396.644, Z    +0.000, E1   -16.434, E3 +332966.886}
SPL {X  -165.650, Y  +410.885, Z    +0.000, E1   -34.864, E3 +332961.984}
SPL {X  -165.650, Y  +448.279, Z    +0.000, E1   -53.294, E3 +332979.829}
SPL {X  -165.650, Y  +465.286, Z    +0.000, E1   -55.209, E3 +332993.680}
SPL {X  -165.650, Y  +513.874, Z    +0.000, E1   -57.683, E3 +333038.489}
ENDSPLINE

SPLINE
SPL {X  -165.650, Y  +513.412, Z    +0.000, E1   -55.245, E3 +333052.084}
SPL {X  -165.650, Y  +495.869, Z    +0.000, E1   -48.812, E3 +333063.386}
ENDSPLINE

SPLINE
SPL {X  -165.650, Y  +502.040, Z    +0.000, E1   -48.856, E3 +333074.130}
SPL {X  -165.650, Y  +507.863, Z    +0.000, E1   -49.013, E3 +333083.550}
SPL {X  -165.650, Y  +512.952, Z    +0.000, E1   -48.898, E3 +333093.327}
SPL {X  -165.650, Y  +519.321, Z    +0.000, E1   -49.041, E3 +333103.795}
SPL {X  -165.650, Y  +524.312, Z    +0.000, E1   -48.855, E3 +333113.820}
SPL {X  -165.650, Y  +532.191, Z    +0.000, E1   -48.944, E3 +333127.488}
SPL {X  -165.650, Y  +541.400, Z    +0.000, E1   -48.945, E3 +333143.862}
SPL {X  -165.650, Y  +548.939, Z    +0.000, E1   -48.968, E3 +333157.040}
SPL {X  -165.650, Y  +553.607, Z    +0.000, E1   -48.716, E3 +333166.858}
SPL {X  -165.650, Y  +562.368, Z    +0.000, E1   -49.014, E3 +333180.918}
SPL {X  -165.650, Y  +570.317, Z    +0.000, E1   -48.893, E3 +333195.661}
SPL {X  -165.650, Y  +577.487, Z    +0.000, E1   -49.001, E3 +333207.769}
SPL {X  -165.650, Y  +581.837, Z    +0.000, E1   -48.612, E3 +333217.802}
SPL {X  -165.650, Y  +588.614, Z    +0.000, E1   -49.053, E3 +333227.320}
SPL {X  -165.650, Y  +593.784, Z    +0.000, E1   -48.711, E3 +333238.606}
SPL {X  -165.650, Y  +600.281, Z    +0.000, E1   -48.957, E3 +333248.708}
SPL {X  -165.650, Y  +606.252, Z    +0.000, E1   -48.984, E3 +333259.241}
SPL {X  -165.650, Y  +612.690, Z    +0.000, E1   -49.044, E3 +333270.270}
SPL {X  -165.650, Y  +617.274, Z    +0.000, E1   -48.670, E3 +333280.719}
SPL {X  -165.650, Y  +624.267, Z    +0.000, E1   -48.953, E3 +333291.531}
SPL {X  -165.650, Y  +632.510, Z    +0.000, E1   -48.976, E3 +333306.286}
SPL {X  -165.650, Y  +641.084, Z    +0.000, E1   -48.892, E3 +333321.928}
SPL {X  -165.650, Y  +648.143, Z    +0.000, E1   -49.033, E3 +333333.597}
SPL {X  -165.650, Y  +655.847, Z    +0.000, E1   -48.917, E3 +333348.215}
SPL {X  -165.650, Y  +663.676, Z    +0.000, E1   -48.809, E3 +333362.653}
SPL {X  -165.650, Y  +669.580, Z    +0.000, E1   -48.844, E3 +333372.991}
SPL {X  -165.650, Y  +675.734, Z    +0.000, E1   -49.021, E3 +333382.898}
SPL {X  -165.552, Y  +681.198, Z    +0.000, E1   -48.804, E3 +333393.978}
SPL {X  -165.221, Y  +687.413, Z    +0.000, E1   -48.790, E3 +333405.150}
SPL {X  -164.785, Y  +692.407, Z    +0.000, E1   -48.653, E3 +333414.865}
SPL {X  -164.074, Y  +698.293, Z    +0.000, E1   -48.857, E3 +333424.149}
SPL {X  -163.489, Y  +702.172, Z    +0.000, E1   -48.443, E3 +333433.466}
SPL {X  -162.217, Y  +709.048, Z    +0.000, E1   -48.328, E3 +333446.606}
SPL {X  -160.800, Y  +715.289, Z    +0.000, E1   -47.964, E3 +333459.613}
SPL {X  -159.392, Y  +720.602, Z    +0.000, E1   -47.892, E3 +333469.525}
SPL {X  -157.947, Y  +725.428, Z    +0.000, E1   -47.498, E3 +333480.264}
SPL {X  -156.133, Y  +730.838, Z    +0.000, E1   -47.305, E3 +333490.981}
SPL {X  -154.870, Y  +734.280, Z    +0.000, E1   -46.924, E3 +333498.985}
SPL {X  -150.529, Y  +744.645, Z    +0.000, E1   -49.720, E3 +333502.258}
SPL {X  -140.987, Y  +762.463, Z    +0.000, E1   -53.922, E3 +333507.290}
SPL {X  -129.526, Y  +778.761, Z    +0.000, E1   -47.396, E3 +333595.353}
ENDSPLINE

SPLINE
SPL {X  -152.848, Y  +739.355, Z    +0.000, E1   -33.672, E3 +333670.922}
SPL {X  -162.700, Y  +706.622, Z    +0.000, E1   -19.657, E3 +333677.079}
SPL {X  -164.822, Y  +692.043, Z    +0.000, E1   -12.043, E3 +333672.717}
SPL {X  -165.501, Y  +682.513, Z    +0.000, E1    -6.586, E3 +333671.412}
SPL {X  -165.650, Y  +674.436, Z    +0.000, E1    -1.443, E3 +333670.187}
SPL {X  -165.650, Y  +670.475, Z    +0.000, E1    +1.794, E3 +333669.848}
SPL {X  -165.650, Y  +667.655, Z    +0.000, E1    +4.420, E3 +333669.644}
SPL {X  -165.650, Y  +664.048, Z    +0.000, E1    +8.230, E3 +333669.021}
SPL {X  -165.650, Y  +658.867, Z    +0.000, E1   +14.313, E3 +333667.485}
SPL {X  -165.650, Y  +650.683, Z    +0.000, E1   +24.801, E3 +333664.920}
SPL {X  -165.650, Y  +636.402, Z    +0.000, E1   +39.824, E3 +333664.883}
SPL {X  -165.650, Y  +586.376, Z    +0.000, E1   +59.481, E3 +333682.555}
SPL {X  -165.650, Y  +554.310, Z    +0.000, E1   +51.914, E3 +333750.599}
ENDSPLINE

SPLINE
SPL {X  -165.650, Y  +561.648, Z    +0.000, E1   +48.058, E3 +333761.416}
ENDSPLINE

SPLINE
SPL {X  -165.650, Y  +556.469, Z    +0.000, E1   +47.823, E3 +333772.284}
SPL {X  -165.650, Y  +549.545, Z    +0.000, E1   +47.953, E3 +333784.410}
SPL {X  -165.650, Y  +544.306, Z    +0.000, E1   +47.619, E3 +333795.968}
SPL {X  -165.650, Y  +537.837, Z    +0.000, E1   +47.880, E3 +333806.494}
SPL {X  -165.650, Y  +530.616, Z    +0.000, E1   +47.886, E3 +333819.860}
SPL {X  -165.650, Y  +524.679, Z    +0.000, E1   +47.721, E3 +333831.752}
SPL {X  -165.650, Y  +517.493, Z    +0.000, E1   +47.895, E3 +333844.130}
SPL {X  -165.650, Y  +511.255, Z    +0.000, E1   +47.920, E3 +333855.419}
SPL {X  -165.650, Y  +507.257, Z    +0.000, E1   +47.748, E3 +333863.801}
SPL {X  -165.650, Y  +501.812, Z    +0.000, E1   +47.738, E3 +333874.084}
SPL {X  -165.650, Y  +493.465, Z    +0.000, E1   +47.959, E3 +333888.255}
SPL {X  -165.650, Y  +486.149, Z    +0.000, E1   +47.831, E3 +333902.530}
SPL {X  -165.650, Y  +479.821, Z    +0.000, E1   +47.727, E3 +333914.804}
SPL {X  -165.650, Y  +472.739, Z    +0.000, E1   +47.923, E3 +333926.823}
SPL {X  -165.650, Y  +465.366, Z    +0.000, E1   +47.775, E3 +333941.402}
SPL {X  -165.650, Y  +457.811, Z    +0.000, E1   +47.987, E3 +333954.019}
SPL {X  -165.650, Y  +451.187, Z    +0.000, E1   +47.917, E3 +333966.763}
SPL {X  -165.650, Y  +439.019, Z    +0.000, E1   +49.830, E3 +333977.085}
SPL {X  -165.650, Y  +435.473, Z    +0.000, E1   +49.263, E3 +333986.806}
SPL {X  -165.650, Y  +428.379, Z    +0.000, E1   +49.373, E3 +333998.578}
SPL {X  -165.650, Y  +423.272, Z    +0.000, E1   +49.176, E3 +334008.714}
SPL {X  -165.650, Y  +416.522, Z    +0.000, E1   +49.338, E3 +334019.692}
SPL {X  -165.650, Y  +410.777, Z    +0.000, E1   +49.173, E3 +334030.744}
SPL {X  -165.650, Y  +402.476, Z    +0.000, E1   +49.356, E3 +334044.430}
SPL {X  -165.650, Y  +393.708, Z    +0.000, E1   +49.252, E3 +334060.421}
SPL {X  -165.650, Y  +386.526, Z    +0.000, E1   +49.193, E3 +334073.366}
SPL {X  -165.650, Y  +381.684, Z    +0.000, E1   +49.061, E3 +334082.651}
SPL {X  -165.602, Y  +374.507, Z    +0.000, E1   +49.269, E3 +334094.243}
SPL {X  -165.255, Y  +367.073, Z    +0.000, E1   +49.394, E3 +334106.435}
SPL {X  -164.828, Y  +362.023, Z    +0.000, E1   +48.964, E3 +334117.951}
SPL {X  -163.908, Y  +354.543, Z    +0.000, E1   +49.169, E3 +334129.899}
SPL {X  -163.052, Y  +349.277, Z    +0.000, E1   +48.680, E3 +334142.005}
SPL {X  -162.125, Y  +344.507, Z    +0.000, E1   +48.543, E3 +334151.144}
SPL {X  -160.947, Y  +339.310, Z    +0.000, E1   +48.561, E3 +334160.253}
SPL {X  -159.860, Y  +335.086, Z    +0.000, E1   +48.145, E3 +334169.965}
SPL {X  -158.277, Y  +329.631, Z    +0.000, E1   +47.981, E3 +334180.587}
SPL {X  -156.804, Y  +325.092, Z    +0.000, E1   +47.609, E3 +334190.480}
SPL {X  -155.465, Y  +321.311, Z    +0.000, E1   +47.446, E3 +334198.015}
SPL {X  -153.706, Y  +316.739, Z    +0.000, E1   +47.523, E3 +334205.628}
SPL {X  -143.727, Y  +296.145, Z    +0.000, E1   +53.260, E3 +334208.772}
SPL {X  -128.440, Y  +273.891, Z    +0.000, E1   +47.966, E3 +334296.018}
ENDSPLINE

SPLINE
SPL {X  -131.798, Y  +278.155, Z    +0.000, E1   +45.574, E3 +334321.645}
SPL {X  -154.181, Y  +317.936, Z    +0.000, E1   +32.662, E3 +334386.981}
SPL {X  -162.537, Y  +346.536, Z    +0.000, E1   +20.123, E3 +334386.202}
SPL {X  -165.197, Y  +366.255, Z    +0.000, E1    +9.700, E3 +334379.997}
SPL {X  -165.621, Y  +375.422, Z    +0.000, E1    +4.067, E3 +334380.398}
SPL {X  -165.650, Y  +379.733, Z    +0.000, E1    +1.160, E3 +334378.704}
SPL {X  -165.650, Y  +383.552, Z    +0.000, E1    -1.868, E3 +334377.954}
SPL {X  -165.650, Y  +388.716, Z    +0.000, E1    -7.003, E3 +334377.358}
SPL {X  -165.650, Y  +396.644, Z    +0.000, E1   -16.434, E3 +334375.977}
SPL {X  -165.650, Y  +410.885, Z    +0.000, E1   -34.864, E3 +334371.075}
SPL {X  -165.650, Y  +448.279, Z    +0.000, E1   -53.294, E3 +334388.920}
SPL {X  -165.650, Y  +465.286, Z    +0.000, E1   -55.209, E3 +334402.771}
SPL {X  -165.650, Y  +513.780, Z    +0.000, E1   -56.183, E3 +334456.288}
ENDSPLINE

SPLINE
SPL {X  -165.650, Y  +495.869, Z    +0.000, E1   -48.812, E3 +334472.477}
ENDSPLINE

SPLINE
SPL {X  -165.650, Y  +502.040, Z    +0.000, E1   -48.856, E3 +334483.220}
SPL {X  -165.650, Y  +507.863, Z    +0.000, E1   -49.013, E3 +334492.640}
SPL {X  -165.650, Y  +512.952, Z    +0.000, E1   -48.898, E3 +334502.418}
SPL {X  -165.650, Y  +519.321, Z    +0.000, E1   -49.041, E3 +334512.886}
SPL {X  -165.650, Y  +524.312, Z    +0.000, E1   -48.855, E3 +334522.911}
SPL {X  -165.650, Y  +532.191, Z    +0.000, E1   -48.944, E3 +334536.579}
SPL {X  -165.650, Y  +541.400, Z    +0.000, E1   -48.945, E3 +334552.953}
SPL {X  -165.650, Y  +548.939, Z    +0.000, E1   -48.968, E3 +334566.131}
SPL {X  -165.650, Y  +553.607, Z    +0.000, E1   -48.716, E3 +334575.949}
SPL {X  -165.650, Y  +562.368, Z    +0.000, E1   -49.014, E3 +334590.009}
SPL {X  -165.650, Y  +570.317, Z    +0.000, E1   -48.893, E3 +334604.752}
SPL {X  -165.650, Y  +577.487, Z    +0.000, E1   -49.001, E3 +334616.860}
SPL {X  -165.650, Y  +581.837, Z    +0.000, E1   -48.612, E3 +334626.893}
SPL {X  -165.650, Y  +588.614, Z    +0.000, E1   -49.053, E3 +334636.411}
SPL {X  -165.650, Y  +593.784, Z    +0.000, E1   -48.711, E3 +334647.696}
SPL {X  -165.650, Y  +600.281, Z    +0.000, E1   -48.957, E3 +334657.799}
SPL {X  -165.650, Y  +606.252, Z    +0.000, E1   -48.984, E3 +334668.332}
SPL {X  -165.650, Y  +612.690, Z    +0.000, E1   -49.044, E3 +334679.361}
SPL {X  -165.650, Y  +617.274, Z    +0.000, E1   -48.670, E3 +334689.810}
SPL {X  -165.650, Y  +624.267, Z    +0.000, E1   -48.953, E3 +334700.622}
SPL {X  -165.650, Y  +632.510, Z    +0.000, E1   -48.976, E3 +334715.377}
SPL {X  -165.650, Y  +641.084, Z    +0.000, E1   -48.892, E3 +334731.019}
SPL {X  -165.650, Y  +648.143, Z    +0.000, E1   -49.033, E3 +334742.688}
SPL {X  -165.650, Y  +655.847, Z    +0.000, E1   -48.917, E3 +334757.306}
SPL {X  -165.650, Y  +663.676, Z    +0.000, E1   -48.809, E3 +334771.744}
SPL {X  -165.650, Y  +669.580, Z    +0.000, E1   -48.844, E3 +334782.082}
SPL {X  -165.650, Y  +675.734, Z    +0.000, E1   -49.021, E3 +334791.989}
SPL {X  -165.552, Y  +681.198, Z    +0.000, E1   -48.804, E3 +334803.069}
SPL {X  -165.221, Y  +687.413, Z    +0.000, E1   -48.790, E3 +334814.240}
SPL {X  -164.785, Y  +692.407, Z    +0.000, E1   -48.653, E3 +334823.956}
SPL {X  -164.074, Y  +698.293, Z    +0.000, E1   -48.857, E3 +334833.240}
SPL {X  -163.489, Y  +702.172, Z    +0.000, E1   -48.443, E3 +334842.557}
SPL {X  -162.217, Y  +709.048, Z    +0.000, E1   -48.328, E3 +334855.696}
SPL {X  -160.800, Y  +715.289, Z    +0.000, E1   -47.964, E3 +334868.704}
SPL {X  -159.392, Y  +720.602, Z    +0.000, E1   -47.892, E3 +334878.616}
SPL {X  -157.947, Y  +725.428, Z    +0.000, E1   -47.498, E3 +334889.355}
SPL {X  -156.133, Y  +730.838, Z    +0.000, E1   -47.305, E3 +334900.072}
SPL {X  -153.862, Y  +736.871, Z    +0.000, E1   -47.425, E3 +334910.059}
SPL {X  -143.211, Y  +758.749, Z    +0.000, E1   -53.445, E3 +334913.702}
SPL {X  -130.133, Y  +777.996, Z    +0.000, E1   -46.969, E3 +335008.805}
ENDSPLINE

SPLINE
SPL {X  -153.839, Y  +736.929, Z    +0.000, E1   -32.772, E3 +335081.876}
SPL {X  -162.700, Y  +706.622, Z    +0.000, E1   -19.657, E3 +335086.170}
SPL {X  -164.822, Y  +692.043, Z    +0.000, E1   -12.043, E3 +335081.808}
SPL {X  -165.501, Y  +682.513, Z    +0.000, E1    -6.586, E3 +335080.503}
SPL {X  -165.650, Y  +674.436, Z    +0.000, E1    -1.443, E3 +335079.278}
SPL {X  -165.650, Y  +669.008, Z    +0.000, E1    +2.993, E3 +335078.833}
SPL {X  -165.650, Y  +663.208, Z    +0.000, E1    +9.118, E3 +335077.917}
SPL {X  -165.650, Y  +657.399, Z    +0.000, E1   +16.251, E3 +335076.036}
SPL {X  -165.650, Y  +650.683, Z    +0.000, E1   +24.801, E3 +335074.011}
SPL {X  -165.650, Y  +636.402, Z    +0.000, E1   +39.824, E3 +335073.974}
SPL {X  -165.650, Y  +586.376, Z    +0.000, E1   +59.481, E3 +335091.646}
SPL {X  -165.650, Y  +558.853, Z    +0.000, E1   +50.142, E3 +335163.116}
SPL {X  -165.650, Y  +558.330, Z    +0.000, E1   +47.867, E3 +335177.829}
SPL {X  -165.650, Y  +549.545, Z    +0.000, E1   +47.953, E3 +335193.501}
SPL {X  -165.650, Y  +541.974, Z    +0.000, E1   +47.882, E3 +335207.890}
SPL {X  -165.650, Y  +535.023, Z    +0.000, E1   +47.697, E3 +335221.879}
SPL {X  -165.650, Y  +526.169, Z    +0.000, E1   +47.853, E3 +335237.474}
SPL {X  -165.650, Y  +517.493, Z    +0.000, E1   +47.895, E3 +335253.221}
SPL {X  -165.650, Y  +509.413, Z    +0.000, E1   +47.884, E3 +335268.300}
SPL {X  -165.650, Y  +501.812, Z    +0.000, E1   +47.738, E3 +335283.175}
SPL {X  -165.650, Y  +493.465, Z    +0.000, E1   +47.959, E3 +335297.346}
SPL {X  -165.650, Y  +486.149, Z    +0.000, E1   +47.831, E3 +335311.621}
SPL {X  -165.650, Y  +477.718, Z    +0.000, E1   +47.870, E3 +335327.060}
SPL {X  -165.650, Y  +469.088, Z    +0.000, E1   +47.982, E3 +335342.280}
SPL {X  -165.650, Y  +464.575, Z    +0.000, E1   +47.451, E3 +335353.694}
SPL {X  -165.650, Y  +457.811, Z    +0.000, E1   +47.987, E3 +335363.110}
SPL {X  -165.650, Y  +451.187, Z    +0.000, E1   +47.917, E3 +335375.854}
SPL {X  -165.650, Y  +437.755, Z    +0.000, E1   +49.519, E3 +335390.420}
ENDSPLINE

SPLINE
SPL {X  -165.650, Y  +443.669, Z    +0.000, E1   +45.313, E3 +335404.384}
ENDSPLINE

SPLINE
SPL {X  -165.650, Y  +436.063, Z    +0.000, E1   +44.972, E3 +335421.970}
SPL {X  -165.650, Y  +427.943, Z    +0.000, E1   +45.362, E3 +335436.008}
SPL {X  -165.650, Y  +422.523, Z    +0.000, E1   +45.103, E3 +335448.686}
SPL {X  -165.650, Y  +415.564, Z    +0.000, E1   +45.195, E3 +335462.225}
SPL {X  -165.650, Y  +410.687, Z    +0.000, E1   +44.955, E3 +335473.541}
SPL {X  -165.650, Y  +402.778, Z    +0.000, E1   +45.323, E3 +335487.622}
SPL {X  -165.650, Y  +396.171, Z    +0.000, E1   +44.969, E3 +335503.043}
SPL {X  -165.650, Y  +390.060, Z    +0.000, E1   +45.007, E3 +335515.276}
SPL {X  -165.650, Y  +383.700, Z    +0.000, E1   +45.345, E3 +335526.200}
SPL {X  -165.650, Y  +379.225, Z    +0.000, E1   +45.073, E3 +335536.889}
SPL {X  -165.591, Y  +374.097, Z    +0.000, E1   +45.069, E3 +335547.370}
SPL {X  -165.372, Y  +368.914, Z    +0.000, E1   +45.103, E3 +335557.730}
SPL {X  -164.987, Y  +363.696, Z    +0.000, E1   +45.006, E3 +335568.953}
SPL {X  -164.256, Y  +357.053, Z    +0.000, E1   +44.969, E3 +335582.756}
SPL {X  -163.441, Y  +351.538, Z    +0.000, E1   +44.749, E3 +335595.119}
SPL {X  -162.419, Y  +345.942, Z    +0.000, E1   +44.540, E3 +335607.851}
SPL {X  -161.210, Y  +340.404, Z    +0.000, E1   +44.250, E3 +335620.676}
SPL {X  -159.961, Y  +335.460, Z    +0.000, E1   +44.205, E3 +335631.039}
SPL {X  -158.595, Y  +330.672, Z    +0.000, E1   +43.797, E3 +335643.017}
SPL {X  -156.695, Y  +324.773, Z    +0.000, E1   +43.987, E3 +335653.914}
SPL {X  -148.318, Y  +304.733, Z    +0.000, E1   +49.897, E3 +335659.150}
SPL {X  -137.641, Y  +286.333, Z    +0.000, E1   +45.396, E3 +335734.010}
SPL {X  -137.518, Y  +286.149, Z    +0.000, E1   +42.648, E3 +335806.519}
ENDSPLINE

SPLINE
SPL {X  -156.430, Y  +324.005, Z    +0.000, E1   +29.926, E3 +335811.654}
SPL {X  -161.387, Y  +341.161, Z    +0.000, E1   +22.590, E3 +335827.496}
SPL {X  -164.566, Y  +359.576, Z    +0.000, E1   +13.425, E3 +335806.089}
SPL {X  -165.355, Y  +368.611, Z    +0.000, E1    +8.407, E3 +335809.670}
SPL {X  -165.614, Y  +375.050, Z    +0.000, E1    +4.520, E3 +335810.974}
SPL {X  -165.650, Y  +379.847, Z    +0.000, E1    +1.364, E3 +335809.323}
SPL {X  -165.650, Y  +383.246, Z    +0.000, E1    -1.216, E3 +335808.417}
SPL {X  -165.650, Y  +386.866, Z    +0.000, E1    -4.337, E3 +335808.469}
SPL {X  -165.650, Y  +394.200, Z    +0.000, E1   -11.943, E3 +335806.236}
SPL {X  -165.650, Y  +405.401, Z    +0.000, E1   -24.512, E3 +335806.056}
SPL {X  -165.650, Y  +418.038, Z    +0.000, E1   -38.688, E3 +335802.284}
SPL {X  -165.650, Y  +461.620, Z    +0.000, E1   -55.594, E3 +335822.462}
SPL {X  -165.650, Y  +505.847, Z    +0.000, E1   -55.467, E3 +335874.435}
ENDSPLINE

SPLINE
SPL {X  -165.650, Y  +495.538, Z    +0.000, E1   -50.621, E3 +335886.919}
SPL {X  -165.650, Y  +484.983, Z    +0.000, E1   -45.406, E3 +335898.990}
ENDSPLINE

SPLINE
SPL {X  -165.650, Y  +492.090, Z    +0.000, E1   -45.292, E3 +335914.013}
SPL {X  -165.650, Y  +498.857, Z    +0.000, E1   -45.339, E3 +335927.350}
SPL {X  -165.650, Y  +505.115, Z    +0.000, E1   -45.299, E3 +335940.298}
SPL {X  -165.650, Y  +510.931, Z    +0.000, E1   -45.250, E3 +335952.289}
SPL {X  -165.650, Y  +516.157, Z    +0.000, E1   -45.240, E3 +335962.963}
SPL {X  -165.650, Y  +521.049, Z    +0.000, E1   -45.236, E3 +335972.916}
SPL {X  -165.650, Y  +527.050, Z    +0.000, E1   -45.345, E3 +335984.412}
SPL {X  -165.650, Y  +532.042, Z    +0.000, E1   -45.233, E3 +335995.156}
SPL {X  -165.650, Y  +537.290, Z    +0.000, E1   -45.204, E3 +336005.996}
SPL {X  -165.650, Y  +544.196, Z    +0.000, E1   -45.432, E3 +336018.671}
SPL {X  -165.650, Y  +548.678, Z    +0.000, E1   -45.162, E3 +336029.234}
SPL {X  -165.650, Y  +554.600, Z    +0.000, E1   -45.345, E3 +336040.211}
SPL {X  -165.650, Y  +561.799, Z    +0.000, E1   -45.312, E3 +336055.080}
SPL {X  -165.650, Y  +567.835, Z    +0.000, E1   -45.186, E3 +336067.887}
SPL {X  -165.650, Y  +573.074, Z    +0.000, E1   -45.379, E3 +336077.378}
SPL {X  -165.650, Y  +579.360, Z    +0.000, E1   -45.300, E3 +336090.663}
SPL {X  -165.650, Y  +584.577, Z    +0.000, E1   -45.167, E3 +336101.886}
SPL {X  -165.650, Y  +590.060, Z    +0.000, E1   -45.221, E3 +336112.777}
SPL {X  -165.650, Y  +596.611, Z    +0.000, E1   -45.390, E3 +336125.013}
SPL {X  -165.650, Y  +603.637, Z    +0.000, E1   -45.296, E3 +336139.932}
SPL {X  -165.650, Y  +610.850, Z    +0.000, E1   -45.208, E3 +336154.940}
SPL {X  -165.650, Y  +617.450, Z    +0.000, E1   -45.402, E3 +336167.143}
SPL {X  -165.650, Y  +622.720, Z    +0.000, E1   -45.272, E3 +336178.540}
SPL {X  -165.650, Y  +627.828, Z    +0.000, E1   -45.174, E3 +336189.497}
SPL {X  -165.650, Y  +634.620, Z    +0.000, E1   -45.438, E3 +336201.703}
SPL {X  -165.650, Y  +640.808, Z    +0.000, E1   -45.294, E3 +336215.077}
SPL {X  -165.650, Y  +646.552, Z    +0.000, E1   -45.137, E3 +336227.601}
SPL {X  -165.650, Y  +652.431, Z    +0.000, E1   -45.333, E3 +336238.356}
SPL {X  -165.650, Y  +657.443, Z    +0.000, E1   -45.316, E3 +336248.612}
SPL {X  -165.650, Y  +662.999, Z    +0.000, E1   -45.214, E3 +336260.484}
SPL {X  -165.650, Y  +668.737, Z    +0.000, E1   -45.236, E3 +336271.999}
SPL {X  -165.650, Y  +675.226, Z    +0.000, E1   -45.503, E3 +336283.503}
SPL {X  -165.597, Y  +679.672, Z    +0.000, E1   -45.206, E3 +336294.224}
SPL {X  -165.388, Y  +684.808, Z    +0.000, E1   -45.192, E3 +336304.731}
SPL {X  -165.020, Y  +689.938, Z    +0.000, E1   -45.107, E3 +336315.674}
SPL {X  -164.358, Y  +696.147, Z    +0.000, E1   -45.160, E3 +336327.940}
SPL {X  -163.631, Y  +701.286, Z    +0.000, E1   -44.994, E3 +336339.232}
SPL {X  -163.047, Y  +704.748, Z    +0.000, E1   -44.682, E3 +336348.056}
SPL {X  -161.884, Y  +710.619, Z    +0.000, E1   -44.738, E3 +336359.681}
SPL {X  -160.692, Y  +715.726, Z    +0.000, E1   -44.379, E3 +336372.003}
SPL {X  -159.384, Y  +720.631, Z    +0.000, E1   -44.155, E3 +336383.153}
SPL {X  -158.321, Y  +724.227, Z    +0.000, E1   -43.955, E3 +336391.474}
SPL {X  -156.604, Y  +729.490, Z    +0.000, E1   -44.229, E3 +336400.641}
SPL {X  -147.100, Y  +751.668, Z    +0.000, E1   -50.624, E3 +336406.528}
SPL {X  -144.116, Y  +757.172, Z    +0.000, E1   -42.809, E3 +336475.924}
SPL {X  -127.227, Y  +781.582, Z    +0.000, E1   -46.780, E3 +336521.594}
ENDSPLINE

SPLINE
SPL {X  -133.736, Y  +773.248, Z    +0.000, E1   -45.385, E3 +336599.636}
SPL {X  -160.761, Y  +715.447, Z    +0.000, E1   -23.748, E3 +336556.486}
SPL {X  -164.304, Y  +696.571, Z    +0.000, E1   -14.525, E3 +336561.710}
SPL {X  -165.374, Y  +685.052, Z    +0.000, E1    -8.166, E3 +336561.103}
SPL {X  -165.648, Y  +676.230, Z    +0.000, E1    -2.814, E3 +336560.254}
SPL {X  -165.650, Y  +670.481, Z    +0.000, E1    +1.454, E3 +336559.184}
SPL {X  -165.650, Y  +665.304, Z    +0.000, E1    +6.303, E3 +336557.686}
SPL {X  -165.650, Y  +660.688, Z    +0.000, E1   +11.392, E3 +336556.819}
SPL {X  -165.650, Y  +655.692, Z    +0.000, E1   +17.061, E3 +336556.241}
SPL {X  -165.650, Y  +646.511, Z    +0.000, E1   +26.434, E3 +336559.022}
SPL {X  -165.650, Y  +637.905, Z    +0.000, E1   +40.225, E3 +336547.146}
SPL {X  -165.650, Y  +607.385, Z    +0.000, E1   +51.775, E3 +336566.904}
SPL {X  -165.650, Y  +598.058, Z    +0.000, E1   +51.157, E3 +336580.366}
SPL {X  -165.650, Y  +553.219, Z    +0.000, E1   +52.865, E3 +336634.548}
ENDSPLINE

SPLINE
SPL {X  -165.650, Y  +569.883, Z    +0.000, E1   +45.183, E3 +336650.225}
ENDSPLINE

